	UF : 0, UT : 6,		CONFIG : 'N U T, 0, 0, 0',
	X =  237.113  mm,	Y =   -360.782  mm,	Z =   -247.837  mm,
	W =  90.000 deg,	P =   -89.765 deg,	R =   30.000 deg
};
P[393]{
   GP1:
	UF : 0, UT : 6,		CONFIG : 'N U T, 0, 0, 0',
	X =  236.281  mm,	Y =   -361.266  mm,	Z =   -247.891  mm,
	W =  90.000 deg,	P =   -89.765 deg,	R =   30.000 deg
};
P[394]{
   GP1:
	UF : 0, UT : 6,		CONFIG : 'N U T, 0, 0, 0',
	X =  236.253  mm,	Y =   -361.209  mm,	Z =   -246.975  mm,
	W =  90.000 deg,	P =   -89.765 deg,	R =   30.000 deg
};
P[395]{
   GP1:
	UF : 0, UT : 6,		CONFIG : 'N U T, 0, 0, 0',
	X =  235.670  mm,	Y =   -361.621  mm,	Z =   -247.913  mm,
	W =  90.000 deg,	P =   -89.765 deg,	R =   30.000 deg
};
P[396]{
   GP1:
	UF : 0, UT : 6,		CONFIG : 'N U T, 0, 0, 0',
	X =  235.399  mm,	Y =   -361.776  mm,	Z =   -247.895  mm,
	W =  90.000 deg,	P =   -89.765 deg,	R =   30.000 deg
};
P[397]{
   GP1:
	UF : 0, UT : 6,		CONFIG : 'N U T, 0, 0, 0',
	X =  234.392  mm,	Y =   -360.505  mm,	Z =   -224.946  mm,
	W =  90.000 deg,	P =   -89.765 deg,	R =   30.000 deg
};
P[398]{
   GP1:
	UF : 0, UT : 6,		CONFIG : 'N U T, 0, 0, 0',
	X =  234.357  mm,	Y =   -360.593  mm,	Z =   -225.785  mm,
	W =  90.000 deg,	P =   -89.765 deg,	R =   30.000 deg
};
P[399]{
   GP1:
	UF : 0, UT : 6,		CONFIG : 'N U T, 0, 0, 0',
	X =  234.000  mm,	Y =   -360.802  mm,	Z =   -225.822  mm,
	W =  90.000 deg,	P =   -89.765 deg,	R =   30.000 deg
};
P[400]{
   GP1:
	UF : 0, UT : 6,		CONFIG : 'N U T, 0, 0, 0',
	X =  233.702  mm,	Y =   -360.970  mm,	Z =   -225.770  mm,
	W =  90.000 deg,	P =   -89.765 deg,	R =   30.000 deg
};
P[401]{
   GP1:
	UF : 0, UT : 6,		CONFIG : 'N U T, 0, 0, 0',
	X =  233.487  mm,	Y =   -361.098  mm,	Z =   -225.822  mm,
	W =  90.000 deg,	P =   -89.765 deg,	R =   30.000 deg
};
P[402]{
   GP1:
	UF : 0, UT : 6,		CONFIG : 'N U T, 0, 0, 0',
	X =  233.404  mm,	Y =   -361.075  mm,	Z =   -224.940  mm,
	W =  90.000 deg,	P =   -89.765 deg,	R =   30.000 deg
};
P[403]{
   GP1:
	UF : 0, UT : 6,		CONFIG : 'N U T, 0, 0, 0',
	X =  232.811  mm,	Y =   -361.483  mm,	Z =   -225.762  mm,
	W =  90.000 deg,	P =   -89.765 deg,	R =   30.000 deg
};
P[404]{
   GP1:
	UF : 0, UT : 6,		CONFIG : 'N U T, 0, 0, 0',
	X =  232.580  mm,	Y =   -361.587  mm,	Z =   -225.392  mm,
	W =  90.000 deg,	P =   -89.765 deg,	R =   30.000 deg
};
P[405]{
   GP1:
	UF : 0, UT : 6,		CONFIG : 'N U T, 0, 0, 0',
	X =  232.529  mm,	Y =   -361.658  mm,	Z =   -225.909  mm,
	W =  90.000 deg,	P =   -89.765 deg,	R =   30.000 deg
};
P[406]{
   GP1:
	UF : 0, UT : 6,		CONFIG : 'N U T, 0, 0, 0',
	X =  232.294  mm,	Y =   -361.754  mm,	Z =   -225.413  mm,
	W =  90.000 deg,	P =   -89.765 deg,	R =   30.000 deg
};
P[407]{
   GP1:
	UF : 0, UT : 6,		CONFIG : 'N U T, 0, 0, 0',
	X =  232.210  mm,	Y =   -361.841  mm,	Z =   -225.896  mm,
	W =  90.000 deg,	P =   -89.765 deg,	R =   30.000 deg
};
P[408]{
   GP1:
	UF : 0, UT : 6,		CONFIG : 'N U T, 0, 0, 0',
	X =  231.623  mm,	Y =   -362.182  mm,	Z =   -225.911  mm,
	W =  90.000 deg,	P =   -89.765 deg,	R =   30.000 deg
};
P[409]{
   GP1:
	UF : 0, UT : 6,		CONFIG : 'N U T, 0, 0, 0',
	X =  231.557  mm,	Y =   -362.142  mm,	Z =   -224.952  mm,
	W =  90.000 deg,	P =   -89.765 deg,	R =   30.000 deg
};
P[410]{
   GP1:
	UF : 0, UT : 6,		CONFIG : 'N U T, 0, 0, 0',
	X =  231.491  mm,	Y =   -362.215  mm,	Z =   -225.396  mm,
	W =  90.000 deg,	P =   -89.765 deg,	R =   30.000 deg
};
P[411]{
   GP1:
	UF : 0, UT : 6,		CONFIG : 'N U T, 0, 0, 0',
	X =  231.269  mm,	Y =   -362.315  mm,	Z =   -225.031  mm,
	W =  90.000 deg,	P =   -89.765 deg,	R =   30.000 deg
};
P[412]{
   GP1:
	UF : 0, UT : 6,		CONFIG : 'N U T, 0, 0, 0',
	X =  231.297  mm,	Y =   -362.369  mm,	Z =   -225.901  mm,
	W =  90.000 deg,	P =   -89.765 deg,	R =   30.000 deg
};
P[413]{
   GP1:
	UF : 0, UT : 6,		CONFIG : 'N U T, 0, 0, 0',
	X =  230.990  mm,	Y =   -362.547  mm,	Z =   -225.923  mm,
	W =  90.000 deg,	P =   -89.765 deg,	R =   30.000 deg
};
P[414]{
   GP1:
	UF : 0, UT : 6,		CONFIG : 'N U T, 0, 0, 0',
	X =  230.655  mm,	Y =   -362.675  mm,	Z =   -225.107  mm,
	W =  90.000 deg,	P =   -89.765 deg,	R =   30.000 deg
};
P[415]{
   GP1:
	UF : 0, UT : 6,		CONFIG : 'N U T, 0, 0, 0',
	X =  230.373  mm,	Y =   -362.893  mm,	Z =   -225.776  mm,
	W =  90.000 deg,	P =   -89.765 deg,	R =   30.000 deg
};
P[416]{
   GP1:
	UF : 0, UT : 6,		CONFIG : 'N U T, 0, 0, 0',
	X =  229.910  mm,	Y =   -363.127  mm,	Z =   -225.378  mm,
	W =  90.000 deg,	P =   -89.765 deg,	R =   30.000 deg
};
P[417]{
   GP1:
	UF : 0, UT : 6,		CONFIG : 'N U T, 0, 0, 0',
	X =  229.140  mm,	Y =   -363.606  mm,	Z =   -225.794  mm,
	W =  90.000 deg,	P =   -89.765 deg,	R =   30.000 deg
};
P[418]{
   GP1:
	UF : 0, UT : 6,		CONFIG : 'N U T, 0, 0, 0',
	X =  228.874  mm,	Y =   -363.726  mm,	Z =   -225.370  mm,
	W =  90.000 deg,	P =   -89.765 deg,	R =   30.000 deg
};
P[419]{
   GP1:
	UF : 0, UT : 6,		CONFIG : 'N U T, 0, 0, 0',
	X =  228.845  mm,	Y =   -363.780  mm,	Z =   -225.848  mm,
	W =  90.000 deg,	P =   -89.765 deg,	R =   30.000 deg
};
P[420]{
   GP1:
	UF : 0, UT : 6,		CONFIG : 'N U T, 0, 0, 0',
	X =  227.859  mm,	Y =   -364.284  mm,	Z =   -225.040  mm,
	W =  90.000 deg,	P =   -89.765 deg,	R =   30.000 deg
};
P[421]{
   GP1:
	UF : 0, UT : 6,		CONFIG : 'N U T, 0, 0, 0',
	X =  227.784  mm,	Y =   -364.357  mm,	Z =   -225.398  mm,
	W =  90.000 deg,	P =   -89.765 deg,	R =   30.000 deg
};
P[422]{
   GP1:
	UF : 0, UT : 6,		CONFIG : 'N U T, 0, 0, 0',
	X =  227.246  mm,	Y =   -364.630  mm,	Z =   -224.931  mm,
	W =  90.000 deg,	P =   -89.765 deg,	R =   30.000 deg
};
P[423]{
   GP1:
	UF : 0, UT : 6,		CONFIG : 'N U T, 0, 0, 0',
	X =  227.248  mm,	Y =   -364.668  mm,	Z =   -225.413  mm,
	W =  90.000 deg,	P =   -89.765 deg,	R =   30.000 deg
};
P[424]{
   GP1:
	UF : 0, UT : 6,		CONFIG : 'N U T, 0, 0, 0',
	X =  226.957  mm,	Y =   -364.870  mm,	Z =   -225.849  mm,
	W =  90.000 deg,	P =   -89.765 deg,	R =   30.000 deg
};
P[425]{
   GP1:
	UF : 0, UT : 6,		CONFIG : 'N U T, 0, 0, 0',
	X =  226.306  mm,	Y =   -365.173  mm,	Z =   -224.949  mm,
	W =  90.000 deg,	P =   -89.765 deg,	R =   30.000 deg
};
P[426]{
   GP1:
	UF : 0, UT : 6,		CONFIG : 'N U T, 0, 0, 0',
	X =  226.123  mm,	Y =   -365.346  mm,	Z =   -225.786  mm,
	W =  90.000 deg,	P =   -89.765 deg,	R =   30.000 deg
};
P[427]{
   GP1:
	UF : 0, UT : 6,		CONFIG : 'N U T, 0, 0, 0',
	X =  225.718  mm,	Y =   -365.520  mm,	Z =   -225.031  mm,
	W =  90.000 deg,	P =   -89.765 deg,	R =   30.000 deg
};
P[428]{
   GP1:
	UF : 0, UT : 6,		CONFIG : 'N U T, 0, 0, 0',
	X =  225.480  mm,	Y =   -365.726  mm,	Z =   -225.890  mm,
	W =  90.000 deg,	P =   -89.765 deg,	R =   30.000 deg
};
P[429]{
   GP1:
	UF : 0, UT : 6,		CONFIG : 'N U T, 0, 0, 0',
	X =  225.376  mm,	Y =   -365.713  mm,	Z =   -224.981  mm,
	W =  90.000 deg,	P =   -89.765 deg,	R =   30.000 deg
};
P[430]{
   GP1:
	UF : 0, UT : 6,		CONFIG : 'N U T, 0, 0, 0',
	X =  225.172  mm,	Y =   -365.903  mm,	Z =   -225.869  mm,
	W =  90.000 deg,	P =   -89.765 deg,	R =   30.000 deg
};
P[431]{
   GP1:
	UF : 0, UT : 6,		CONFIG : 'N U T, 0, 0, 0',
	X =  224.799  mm,	Y =   -366.046  mm,	Z =   -224.974  mm,
	W =  90.000 deg,	P =   -89.765 deg,	R =   30.000 deg
};
P[432]{
   GP1:
	UF : 0, UT : 6,		CONFIG : 'N U T, 0, 0, 0',
	X =  224.881  mm,	Y =   -366.070  mm,	Z =   -225.869  mm,
	W =  90.000 deg,	P =   -89.765 deg,	R =   30.000 deg
};
P[433]{
   GP1:
	UF : 0, UT : 6,		CONFIG : 'N U T, 0, 0, 0',
	X =  224.484  mm,	Y =   -366.225  mm,	Z =   -224.935  mm,
	W =  90.000 deg,	P =   -89.765 deg,	R =   30.000 deg
};
P[434]{
   GP1:
	UF : 0, UT : 6,		CONFIG : 'N U T, 0, 0, 0',
	X =  223.897  mm,	Y =   -366.567  mm,	Z =   -224.985  mm,
	W =  90.000 deg,	P =   -89.765 deg,	R =   30.000 deg
};
P[435]{
   GP1:
	UF : 0, UT : 6,		CONFIG : 'N U T, 0, 0, 0',
	X =  223.958  mm,	Y =   -366.608  mm,	Z =   -225.921  mm,
	W =  90.000 deg,	P =   -89.765 deg,	R =   30.000 deg
};
P[436]{
   GP1:
	UF : 0, UT : 6,		CONFIG : 'N U T, 0, 0, 0',
	X =  223.659  mm,	Y =   -366.774  mm,	Z =   -225.845  mm,
	W =  90.000 deg,	P =   -89.765 deg,	R =   30.000 deg
};
P[437]{
   GP1:
	UF : 0, UT : 6,		CONFIG : 'N U T, 0, 0, 0',
	X =  223.279  mm,	Y =   -366.933  mm,	Z =   -225.088  mm,
	W =  90.000 deg,	P =   -89.765 deg,	R =   30.000 deg
};
P[438]{
   GP1:
	UF : 0, UT : 6,		CONFIG : 'N U T, 0, 0, 0',
	X =  222.812  mm,	Y =   -367.228  mm,	Z =   -225.404  mm,
	W =  90.000 deg,	P =   -89.765 deg,	R =   30.000 deg
};
P[439]{
   GP1:
	UF : 0, UT : 6,		CONFIG : 'N U T, 0, 0, 0',
	X =  222.634  mm,	Y =   -367.307  mm,	Z =   -225.106  mm,
	W =  90.000 deg,	P =   -89.765 deg,	R =   30.000 deg
};
P[440]{
   GP1:
	UF : 0, UT : 6,		CONFIG : 'N U T, 0, 0, 0',
	X =  222.336  mm,	Y =   -367.475  mm,	Z =   -225.055  mm,
	W =  90.000 deg,	P =   -89.765 deg,	R =   30.000 deg
};
P[441]{
   GP1:
	UF : 0, UT : 6,		CONFIG : 'N U T, 0, 0, 0',
	X =  222.421  mm,	Y =   -367.495  mm,	Z =   -225.924  mm,
	W =  90.000 deg,	P =   -89.765 deg,	R =   30.000 deg
};
P[442]{
   GP1:
	UF : 0, UT : 6,		CONFIG : 'N U T, 0, 0, 0',
	X =  222.156  mm,	Y =   -367.606  mm,	Z =   -225.402  mm,
	W =  90.000 deg,	P =   -89.765 deg,	R =   30.000 deg
};
P[443]{
   GP1:
	UF : 0, UT : 6,		CONFIG : 'N U T, 0, 0, 0',
	X =  222.101  mm,	Y =   -367.678  mm,	Z =   -225.899  mm,
	W =  90.000 deg,	P =   -89.765 deg,	R =   30.000 deg
};
P[444]{
   GP1:
	UF : 0, UT : 6,		CONFIG : 'N U T, 0, 0, 0',
	X =  221.716  mm,	Y =   -367.828  mm,	Z =   -224.998  mm,
	W =  90.000 deg,	P =   -89.765 deg,	R =   30.000 deg
};
P[445]{
   GP1:
	UF : 0, UT : 6,		CONFIG : 'N U T, 0, 0, 0',
	X =  221.807  mm,	Y =   -367.841  mm,	Z =   -225.809  mm,
	W =  90.000 deg,	P =   -89.765 deg,	R =   30.000 deg
};
P[446]{
   GP1:
	UF : 0, UT : 6,		CONFIG : 'N U T, 0, 0, 0',
	X =  221.506  mm,	Y =   -368.013  mm,	Z =   -225.782  mm,
	W =  90.000 deg,	P =   -89.765 deg,	R =   30.000 deg
};
P[447]{
   GP1:
	UF : 0, UT : 6,		CONFIG : 'N U T, 0, 0, 0',
	X =  221.122  mm,	Y =   -368.170  mm,	Z =   -224.979  mm,
	W =  90.000 deg,	P =   -89.765 deg,	R =   30.000 deg
};
P[448]{
   GP1:
	UF : 0, UT : 6,		CONFIG : 'N U T, 0, 0, 0',
	X =  220.843  mm,	Y =   -368.401  mm,	Z =   -225.860  mm,
	W =  90.000 deg,	P =   -89.765 deg,	R =   30.000 deg
};
P[449]{
   GP1:
	UF : 0, UT : 6,		CONFIG : 'N U T, 0, 0, 0',
	X =  220.507  mm,	Y =   -368.525  mm,	Z =   -224.981  mm,
	W =  90.000 deg,	P =   -89.765 deg,	R =   30.000 deg
};
P[450]{
   GP1:
	UF : 0, UT : 6,		CONFIG : 'N U T, 0, 0, 0',
	X =  220.223  mm,	Y =   -368.756  mm,	Z =   -225.819  mm,
	W =  90.000 deg,	P =   -89.765 deg,	R =   30.000 deg
};
P[451]{
   GP1:
	UF : 0, UT : 6,		CONFIG : 'N U T, 0, 0, 0',
	X =  219.902  mm,	Y =   -368.872  mm,	Z =   -224.956  mm,
	W =  90.000 deg,	P =   -89.765 deg,	R =   30.000 deg
};
P[452]{
   GP1:
	UF : 0, UT : 6,		CONFIG : 'N U T, 0, 0, 0',
	X =  219.585  mm,	Y =   -369.089  mm,	Z =   -225.369  mm,
	W =  90.000 deg,	P =   -89.765 deg,	R =   30.000 deg
};
P[453]{
   GP1:
	UF : 0, UT : 6,		CONFIG : 'N U T, 0, 0, 0',
	X =  219.644  mm,	Y =   -369.097  mm,	Z =   -225.904  mm,
	W =  90.000 deg,	P =   -89.765 deg,	R =   30.000 deg
};
P[454]{
   GP1:
	UF : 0, UT : 6,		CONFIG : 'N U T, 0, 0, 0',
	X =  219.320  mm,	Y =   -369.278  mm,	Z =   -225.830  mm,
	W =  90.000 deg,	P =   -89.765 deg,	R =   30.000 deg
};
P[455]{
   GP1:
	UF : 0, UT : 6,		CONFIG : 'N U T, 0, 0, 0',
	X =  218.586  mm,	Y =   -369.630  mm,	Z =   -224.926  mm,
	W =  90.000 deg,	P =   -89.765 deg,	R =   30.000 deg
};
P[456]{
   GP1:
	UF : 0, UT : 6,		CONFIG : 'N U T, 0, 0, 0',
	X =  218.442  mm,	Y =   -369.788  mm,	Z =   -225.856  mm,
	W =  90.000 deg,	P =   -89.765 deg,	R =   30.000 deg
};
P[457]{
   GP1:
	UF : 0, UT : 6,		CONFIG : 'N U T, 0, 0, 0',
	X =  217.955  mm,	Y =   -370.032  mm,	Z =   -225.398  mm,
	W =  90.000 deg,	P =   -89.765 deg,	R =   30.000 deg
};
P[458]{
   GP1:
	UF : 0, UT : 6,		CONFIG : 'N U T, 0, 0, 0',
	X =  217.837  mm,	Y =   -370.100  mm,	Z =   -225.400  mm,
	W =  90.000 deg,	P =   -89.765 deg,	R =   30.000 deg
};
P[459]{
   GP1:
	UF : 0, UT : 6,		CONFIG : 'N U T, 0, 0, 0',
	X =  217.794  mm,	Y =   -370.161  mm,	Z =   -225.844  mm,
	W =  90.000 deg,	P =   -89.765 deg,	R =   30.000 deg
};
P[460]{
   GP1:
	UF : 0, UT : 6,		CONFIG : 'N U T, 0, 0, 0',
	X =  217.511  mm,	Y =   -370.286  mm,	Z =   -225.369  mm,
	W =  90.000 deg,	P =   -89.765 deg,	R =   30.000 deg
};
P[461]{
   GP1:
	UF : 0, UT : 6,		CONFIG : 'N U T, 0, 0, 0',
	X =  217.487  mm,	Y =   -370.338  mm,	Z =   -225.839  mm,
	W =  90.000 deg,	P =   -89.765 deg,	R =   30.000 deg
};
P[462]{
   GP1:
	UF : 0, UT : 6,		CONFIG : 'N U T, 0, 0, 0',
	X =  217.210  mm,	Y =   -370.501  mm,	Z =   -225.878  mm,
	W =  90.000 deg,	P =   -89.765 deg,	R =   30.000 deg
};
P[463]{
   GP1:
	UF : 0, UT : 6,		CONFIG : 'N U T, 0, 0, 0',
	X =  216.778  mm,	Y =   -370.682  mm,	Z =   -225.031  mm,
	W =  90.000 deg,	P =   -89.765 deg,	R =   30.000 deg
};
P[464]{
   GP1:
	UF : 0, UT : 6,		CONFIG : 'N U T, 0, 0, 0',
	X =  216.880  mm,	Y =   -370.686  mm,	Z =   -225.816  mm,
	W =  90.000 deg,	P =   -89.765 deg,	R =   30.000 deg
};
P[465]{
   GP1:
	UF : 0, UT : 6,		CONFIG : 'N U T, 0, 0, 0',
	X =  216.154  mm,	Y =   -371.071  mm,	Z =   -225.383  mm,
	W =  90.000 deg,	P =   -89.765 deg,	R =   30.000 deg
};
P[466]{
   GP1:
	UF : 0, UT : 6,		CONFIG : 'N U T, 0, 0, 0',
	X =  215.904  mm,	Y =   -371.214  mm,	Z =   -225.372  mm,
	W =  90.000 deg,	P =   -89.765 deg,	R =   30.000 deg
};
P[467]{
   GP1:
	UF : 0, UT : 6,		CONFIG : 'N U T, 0, 0, 0',
	X =  215.958  mm,	Y =   -371.227  mm,	Z =   -225.918  mm,
	W =  90.000 deg,	P =   -89.765 deg,	R =   30.000 deg
};
P[468]{
   GP1:
	UF : 0, UT : 6,		CONFIG : 'N U T, 0, 0, 0',
	X =  215.665  mm,	Y =   -371.387  mm,	Z =   -225.804  mm,
	W =  90.000 deg,	P =   -89.765 deg,	R =   30.000 deg
};
P[469]{
   GP1:
	UF : 0, UT : 6,		CONFIG : 'N U T, 0, 0, 0',
	X =  215.331  mm,	Y =   -371.586  mm,	Z =   -225.886  mm,
	W =  90.000 deg,	P =   -89.765 deg,	R =   30.000 deg
};
P[470]{
   GP1:
	UF : 0, UT : 6,		CONFIG : 'N U T, 0, 0, 0',
	X =  215.026  mm,	Y =   -371.742  mm,	Z =   -225.177  mm,
	W =  90.000 deg,	P =   -89.765 deg,	R =   30.000 deg
};
P[471]{
   GP1:
	UF : 0, UT : 6,		CONFIG : 'N U T, 0, 0, 0',
	X =  215.096  mm,	Y =   -371.773  mm,	Z =   -225.898  mm,
	W =  90.000 deg,	P =   -89.765 deg,	R =   30.000 deg
};
P[472]{
   GP1:
	UF : 0, UT : 6,		CONFIG : 'N U T, 0, 0, 0',
	X =  215.157  mm,	Y =   -372.393  mm,	Z =   -224.958  mm,
	W =  90.000 deg,	P =   -89.765 deg,	R =   30.000 deg
};
P[473]{
   GP1:
	UF : 0, UT : 6,		CONFIG : 'N U T, 0, 0, 0',
	X =  215.297  mm,	Y =   -372.394  mm,	Z =   -225.902  mm,
	W =  90.000 deg,	P =   -89.765 deg,	R =   30.000 deg
};
P[474]{
   GP1:
	UF : 0, UT : 6,		CONFIG : 'N U T, 0, 0, 0',
	X =  215.529  mm,	Y =   -372.532  mm,	Z =   -225.806  mm,
	W =  90.000 deg,	P =   -89.765 deg,	R =   30.000 deg
};
P[475]{
   GP1:
	UF : 0, UT : 6,		CONFIG : 'N U T, 0, 0, 0',
	X =  215.945  mm,	Y =   -372.668  mm,	Z =   -225.782  mm,
	W =  90.000 deg,	P =   -89.765 deg,	R =   30.000 deg
};
P[476]{
   GP1:
	UF : 0, UT : 6,		CONFIG : 'N U T, 0, 0, 0',
	X =  187.636  mm,	Y =   -376.299  mm,	Z =   -225.905  mm,
	W =  179.765 deg,	P =   0.000 deg,	R =   30.000 deg
};
P[477]{
   GP1:
	UF : 0, UT : 6,		CONFIG : 'N U T, 0, 0, 0',
	X =  187.516  mm,	Y =   -376.334  mm,	Z =   -225.076  mm,
	W =  179.765 deg,	P =   0.000 deg,	R =   30.000 deg
};
P[478]{
   GP1:
	UF : 0, UT : 6,		CONFIG : 'N U T, 0, 0, 0',
	X =  186.272  mm,	Y =   -378.286  mm,	Z =   -224.926  mm,
	W =  179.765 deg,	P =   0.000 deg,	R =   30.000 deg
};
P[479]{
   GP1:
	UF : 0, UT : 6,		CONFIG : 'N U T, 0, 0, 0',
	X =  186.053  mm,	Y =   -379.156  mm,	Z =   -225.859  mm,
	W =  179.765 deg,	P =   0.000 deg,	R =   30.000 deg
};
P[480]{
   GP1:
	UF : 0, UT : 6,		CONFIG : 'N U T, 0, 0, 0',
	X =  185.851  mm,	Y =   -379.926  mm,	Z =   -225.382  mm,
	W =  179.765 deg,	P =   0.000 deg,	R =   30.000 deg
};
P[481]{
   GP1:
	UF : 0, UT : 6,		CONFIG : 'N U T, 0, 0, 0',
	X =  185.800  mm,	Y =   -380.295  mm,	Z =   -225.483  mm,
	W =  179.765 deg,	P =   0.000 deg,	R =   30.000 deg
};
P[482]{
   GP1:
	UF : 0, UT : 6,		CONFIG : 'N U T, 0, 0, 0',
	X =  185.847  mm,	Y =   -380.797  mm,	Z =   -225.872  mm,
	W =  179.765 deg,	P =   0.000 deg,	R =   30.000 deg
};
P[483]{
   GP1:
	UF : 0, UT : 6,		CONFIG : 'N U T, 0, 0, 0',
	X =  185.769  mm,	Y =   -380.859  mm,	Z =   -224.974  mm,
	W =  179.765 deg,	P =   0.000 deg,	R =   30.000 deg
};
P[484]{
   GP1:
	UF : 0, UT : 6,		CONFIG : 'N U T, 0, 0, 0',
	X =  185.896  mm,	Y =   -381.491  mm,	Z =   -225.879  mm,
	W =  179.765 deg,	P =   0.000 deg,	R =   30.000 deg
};
P[485]{
   GP1:
	UF : 0, UT : 6,		CONFIG : 'N U T, 0, 0, 0',
	X =  186.008  mm,	Y =   -382.255  mm,	Z =   -225.033  mm,
	W =  179.765 deg,	P =   0.000 deg,	R =   30.000 deg
};
P[486]{
   GP1:
	UF : 0, UT : 6,		CONFIG : 'N U T, 0, 0, 0',
	X =  186.228  mm,	Y =   -382.820  mm,	Z =   -224.959  mm,
	W =  179.765 deg,	P =   0.000 deg,	R =   30.000 deg
};
P[487]{
   GP1:
	UF : 0, UT : 6,		CONFIG : 'N U T, 0, 0, 0',
	X =  186.619  mm,	Y =   -383.588  mm,	Z =   -225.001  mm,
	W =  179.765 deg,	P =   0.000 deg,	R =   30.000 deg
};
P[488]{
   GP1:
	UF : 0, UT : 6,		CONFIG : 'N U T, 0, 0, 0',
	X =  186.703  mm,	Y =   -383.610  mm,	Z =   -225.898  mm,
	W =  179.765 deg,	P =   0.000 deg,	R =   30.000 deg
};
P[489]{
   GP1:
	UF : 0, UT : 6,		CONFIG : 'N U T, 0, 0, 0',
	X =  187.014  mm,	Y =   -384.264  mm,	Z =   -225.061  mm,
	W =  179.765 deg,	P =   0.000 deg,	R =   30.000 deg
};
P[490]{
   GP1:
	UF : 0, UT : 6,		CONFIG : 'N U T, 0, 0, 0',
	X =  187.375  mm,	Y =   -384.782  mm,	Z =   -225.838  mm,
	W =  179.765 deg,	P =   0.000 deg,	R =   30.000 deg
};
P[491]{
   GP1:
	UF : 0, UT : 6,		CONFIG : 'N U T, 0, 0, 0',
	X =  187.642  mm,	Y =   -385.308  mm,	Z =   -225.374  mm,
	W =  179.765 deg,	P =   0.000 deg,	R =   30.000 deg
};
P[492]{
   GP1:
	UF : 0, UT : 6,		CONFIG : 'N U T, 0, 0, 0',
	X =  188.498  mm,	Y =   -386.785  mm,	Z =   -225.413  mm,
	W =  179.765 deg,	P =   0.000 deg,	R =   30.000 deg
};
P[493]{
   GP1:
	UF : 0, UT : 6,		CONFIG : 'N U T, 0, 0, 0',
	X =  188.473  mm,	Y =   -386.803  mm,	Z =   -224.982  mm,
	W =  179.765 deg,	P =   0.000 deg,	R =   30.000 deg
};
P[494]{
   GP1:
	UF : 0, UT : 6,		CONFIG : 'N U T, 0, 0, 0',
	X =  188.877  mm,	Y =   -387.392  mm,	Z =   -225.780  mm,
	W =  179.765 deg,	P =   0.000 deg,	R =   30.000 deg
};
P[495]{
   GP1:
	UF : 0, UT : 6,		CONFIG : 'N U T, 0, 0, 0',
	X =  189.626  mm,	Y =   -388.676  mm,	Z =   -225.866  mm,
	W =  179.765 deg,	P =   0.000 deg,	R =   30.000 deg
};
P[496]{
   GP1:
	UF : 0, UT : 6,		CONFIG : 'N U T, 0, 0, 0',
	X =  190.032  mm,	Y =   -389.448  mm,	Z =   -225.376  mm,
	W =  179.765 deg,	P =   0.000 deg,	R =   30.000 deg
};
P[497]{
   GP1:
	UF : 0, UT : 6,		CONFIG : 'N U T, 0, 0, 0',
	X =  190.306  mm,	Y =   -389.869  mm,	Z =   -225.756  mm,
	W =  179.765 deg,	P =   0.000 deg,	R =   30.000 deg
};
P[498]{
   GP1:
	UF : 0, UT : 6,		CONFIG : 'N U T, 0, 0, 0',
	X =  191.062  mm,	Y =   -391.232  mm,	Z =   -225.376  mm,
	W =  179.765 deg,	P =   0.000 deg,	R =   30.000 deg
};
P[499]{
   GP1:
	UF : 0, UT : 6,		CONFIG : 'N U T, 0, 0, 0',
	X =  191.772  mm,	Y =   -392.386  mm,	Z =   -225.912  mm,
	W =  179.765 deg,	P =   0.000 deg,	R =   30.000 deg
};
P[500]{
   GP1:
	UF : 0, UT : 6,		CONFIG : 'N U T, 0, 0, 0',
	X =  191.716  mm,	Y =   -392.426  mm,	Z =   -224.935  mm,
	W =  179.765 deg,	P =   0.000 deg,	R =   30.000 deg
};
P[501]{
   GP1:
	UF : 0, UT : 6,		CONFIG : 'N U T, 0, 0, 0',
	X =  192.126  mm,	Y =   -393.072  mm,	Z =   -225.383  mm,
	W =  179.765 deg,	P =   0.000 deg,	R =   30.000 deg
};
P[502]{
   GP1:
	UF : 0, UT : 6,		CONFIG : 'N U T, 0, 0, 0',
	X =  192.449  mm,	Y =   -393.561  mm,	Z =   -225.890  mm,
	W =  179.765 deg,	P =   0.000 deg,	R =   30.000 deg
};
P[503]{
   GP1:
	UF : 0, UT : 6,		CONFIG : 'N U T, 0, 0, 0',
	X =  192.468  mm,	Y =   -393.712  mm,	Z =   -225.051  mm,
	W =  179.765 deg,	P =   0.000 deg,	R =   30.000 deg
};
P[504]{
   GP1:
	UF : 0, UT : 6,		CONFIG : 'N U T, 0, 0, 0',
	X =  193.110  mm,	Y =   -394.836  mm,	Z =   -224.967  mm,
	W =  179.765 deg,	P =   0.000 deg,	R =   30.000 deg
};
P[505]{
   GP1:
	UF : 0, UT : 6,		CONFIG : 'N U T, 0, 0, 0',
	X =  193.212  mm,	Y =   -394.888  mm,	Z =   -225.862  mm,
	W =  179.765 deg,	P =   0.000 deg,	R =   30.000 deg
};
P[506]{
   GP1:
	UF : 0, UT : 6,		CONFIG : 'N U T, 0, 0, 0',
	X =  193.527  mm,	Y =   -395.560  mm,	Z =   -224.953  mm,
	W =  179.765 deg,	P =   0.000 deg,	R =   30.000 deg
};
P[507]{
   GP1:
	UF : 0, UT : 6,		CONFIG : 'N U T, 0, 0, 0',
	X =  194.305  mm,	Y =   -396.776  mm,	Z =   -225.891  mm,
	W =  179.765 deg,	P =   0.000 deg,	R =   30.000 deg
};
P[508]{
   GP1:
	UF : 0, UT : 6,		CONFIG : 'N U T, 0, 0, 0',
	X =  194.425  mm,	Y =   -397.052  mm,	Z =   -225.405  mm,
	W =  179.765 deg,	P =   0.000 deg,	R =   30.000 deg
};
P[509]{
   GP1:
	UF : 0, UT : 6,		CONFIG : 'N U T, 0, 0, 0',
	X =  194.620  mm,	Y =   -397.452  mm,	Z =   -224.964  mm,
	W =  179.765 deg,	P =   0.000 deg,	R =   30.000 deg
};
P[510]{
   GP1:
	UF : 0, UT : 6,		CONFIG : 'N U T, 0, 0, 0',
	X =  194.695  mm,	Y =   -397.452  mm,	Z =   -225.885  mm,
	W =  179.765 deg,	P =   0.000 deg,	R =   30.000 deg
};
P[511]{
   GP1:
	UF : 0, UT : 6,		CONFIG : 'N U T, 0, 0, 0',
	X =  194.972  mm,	Y =   -398.059  mm,	Z =   -224.972  mm,
	W =  179.765 deg,	P =   0.000 deg,	R =   30.000 deg
};
P[512]{
   GP1:
	UF : 0, UT : 6,		CONFIG : 'N U T, 0, 0, 0',
	X =  195.239  mm,	Y =   -398.464  mm,	Z =   -225.395  mm,
	W =  179.765 deg,	P =   0.000 deg,	R =   30.000 deg
};
P[513]{
   GP1:
	UF : 0, UT : 6,		CONFIG : 'N U T, 0, 0, 0',
	X =  195.836  mm,	Y =   -399.432  mm,	Z =   -225.860  mm,
	W =  179.765 deg,	P =   0.000 deg,	R =   30.000 deg
};
P[514]{
   GP1:
	UF : 0, UT : 6,		CONFIG : 'N U T, 0, 0, 0',
	X =  195.979  mm,	Y =   -399.749  mm,	Z =   -225.363  mm,
	W =  179.765 deg,	P =   0.000 deg,	R =   30.000 deg
};
P[515]{
   GP1:
	UF : 0, UT : 6,		CONFIG : 'N U T, 0, 0, 0',
	X =  196.097  mm,	Y =   -400.011  mm,	Z =   -224.947  mm,
	W =  179.765 deg,	P =   0.000 deg,	R =   30.000 deg
};
P[516]{
   GP1:
	UF : 0, UT : 6,		CONFIG : 'N U T, 0, 0, 0',
	X =  196.178  mm,	Y =   -400.041  mm,	Z =   -225.740  mm,
	W =  179.765 deg,	P =   0.000 deg,	R =   30.000 deg
};
P[517]{
   GP1:
	UF : 0, UT : 6,		CONFIG : 'N U T, 0, 0, 0',
	X =  196.456  mm,	Y =   -400.527  mm,	Z =   -225.708  mm,
	W =  179.765 deg,	P =   0.000 deg,	R =   30.000 deg
};
P[518]{
   GP1:
	UF : 0, UT : 6,		CONFIG : 'N U T, 0, 0, 0',
	X =  196.993  mm,	Y =   -401.498  mm,	Z =   -225.413  mm,
	W =  179.765 deg,	P =   0.000 deg,	R =   30.000 deg
};
P[519]{
   GP1:
	UF : 0, UT : 6,		CONFIG : 'N U T, 0, 0, 0',
	X =  197.525  mm,	Y =   -402.479  mm,	Z =   -225.000  mm,
	W =  179.765 deg,	P =   0.000 deg,	R =   30.000 deg
};
P[520]{
   GP1:
	UF : 0, UT : 6,		CONFIG : 'N U T, 0, 0, 0',
	X =  197.618  mm,	Y =   -402.582  mm,	Z =   -225.399  mm,
	W =  179.765 deg,	P =   0.000 deg,	R =   30.000 deg
};
P[521]{
   GP1:
	UF : 0, UT : 6,		CONFIG : 'N U T, 0, 0, 0',
	X =  197.819  mm,	Y =   -402.997  mm,	Z =   -224.930  mm,
	W =  179.765 deg,	P =   0.000 deg,	R =   30.000 deg
};
P[522]{
   GP1:
	UF : 0, UT : 6,		CONFIG : 'N U T, 0, 0, 0',
	X =  198.007  mm,	Y =   -403.202  mm,	Z =   -225.792  mm,
	W =  179.765 deg,	P =   0.000 deg,	R =   30.000 deg
};
P[523]{
   GP1:
	UF : 0, UT : 6,		CONFIG : 'N U T, 0, 0, 0',
	X =  198.357  mm,	Y =   -403.809  mm,	Z =   -225.778  mm,
	W =  179.765 deg,	P =   0.000 deg,	R =   30.000 deg
};
P[524]{
   GP1:
	UF : 0, UT : 6,		CONFIG : 'N U T, 0, 0, 0',
	X =  198.596  mm,	Y =   -404.332  mm,	Z =   -225.007  mm,
	W =  179.765 deg,	P =   0.000 deg,	R =   30.000 deg
};
P[525]{
   GP1:
	UF : 0, UT : 6,		CONFIG : 'N U T, 0, 0, 0',
	X =  198.663  mm,	Y =   -404.328  mm,	Z =   -225.859  mm,
	W =  179.765 deg,	P =   0.000 deg,	R =   30.000 deg
};
P[526]{
   GP1:
	UF : 0, UT : 6,		CONFIG : 'N U T, 0, 0, 0',
	X =  199.022  mm,	Y =   -405.057  mm,	Z =   -225.090  mm,
	W =  179.765 deg,	P =   0.000 deg,	R =   30.000 deg
};
P[527]{
   GP1:
	UF : 0, UT : 6,		CONFIG : 'N U T, 0, 0, 0',
	X =  199.160  mm,	Y =   -405.255  mm,	Z =   -225.389  mm,
	W =  179.765 deg,	P =   0.000 deg,	R =   30.000 deg
};
P[528]{
   GP1:
	UF : 0, UT : 6,		CONFIG : 'N U T, 0, 0, 0',
	X =  199.411  mm,	Y =   -405.618  mm,	Z =   -225.906  mm,
	W =  179.765 deg,	P =   0.000 deg,	R =   30.000 deg
};
P[529]{
   GP1:
	UF : 0, UT : 6,		CONFIG : 'N U T, 0, 0, 0',
	X =  199.783  mm,	Y =   -406.278  mm,	Z =   -225.793  mm,
	W =  179.765 deg,	P =   0.000 deg,	R =   30.000 deg
};
P[530]{
   GP1:
	UF : 0, UT : 6,		CONFIG : 'N U T, 0, 0, 0',
	X =  200.163  mm,	Y =   -406.994  mm,	Z =   -225.381  mm,
	W =  179.765 deg,	P =   0.000 deg,	R =   30.000 deg
};
P[531]{
   GP1:
	UF : 0, UT : 6,		CONFIG : 'N U T, 0, 0, 0',
	X =  200.461  mm,	Y =   -407.455  mm,	Z =   -225.770  mm,
	W =  179.765 deg,	P =   0.000 deg,	R =   30.000 deg
};
P[532]{
   GP1:
	UF : 0, UT : 6,		CONFIG : 'N U T, 0, 0, 0',
	X =  200.460  mm,	Y =   -407.564  mm,	Z =   -224.979  mm,
	W =  179.765 deg,	P =   0.000 deg,	R =   30.000 deg
};
P[533]{
   GP1:
	UF : 0, UT : 6,		CONFIG : 'N U T, 0, 0, 0',
	X =  200.697  mm,	Y =   -407.920  mm,	Z =   -225.364  mm,
	W =  179.765 deg,	P =   0.000 deg,	R =   30.000 deg
};
P[534]{
   GP1:
	UF : 0, UT : 6,		CONFIG : 'N U T, 0, 0, 0',
	X =  200.853  mm,	Y =   -408.124  mm,	Z =   -225.829  mm,
	W =  179.765 deg,	P =   0.000 deg,	R =   30.000 deg
};
P[535]{
   GP1:
	UF : 0, UT : 6,		CONFIG : 'N U T, 0, 0, 0',
	X =  201.213  mm,	Y =   -408.809  mm,	Z =   -225.405  mm,
	W =  179.765 deg,	P =   0.000 deg,	R =   30.000 deg
};
P[536]{
   GP1:
	UF : 0, UT : 6,		CONFIG : 'N U T, 0, 0, 0',
	X =  201.559  mm,	Y =   -409.349  mm,	Z =   -225.819  mm,
	W =  179.765 deg,	P =   0.000 deg,	R =   30.000 deg
};
P[537]{
   GP1:
	UF : 0, UT : 6,		CONFIG : 'N U T, 0, 0, 0',
	X =  201.861  mm,	Y =   -409.821  mm,	Z =   -225.925  mm,
	W =  179.765 deg,	P =   0.000 deg,	R =   30.000 deg
};
P[538]{
   GP1:
	UF : 0, UT : 6,		CONFIG : 'N U T, 0, 0, 0',
	X =  201.962  mm,	Y =   -410.061  mm,	Z =   -225.152  mm,
	W =  179.765 deg,	P =   0.000 deg,	R =   30.000 deg
};
P[539]{
   GP1:
	UF : 0, UT : 6,		CONFIG : 'N U T, 0, 0, 0',
	X =  202.367  mm,	Y =   -410.521  mm,	Z =   -225.735  mm,
	W =  179.765 deg,	P =   0.000 deg,	R =   30.000 deg
};
P[540]{
   GP1:
	UF : 0, UT : 6,		CONFIG : 'N U T, 0, 0, 0',
	X =  204.004  mm,	Y =   -411.840  mm,	Z =   -224.989  mm,
	W =  179.765 deg,	P =   0.000 deg,	R =   30.000 deg
};
P[541]{
   GP1:
	UF : 0, UT : 6,		CONFIG : 'N U T, 0, 0, 0',
	X =  204.055  mm,	Y =   -411.791  mm,	Z =   -225.781  mm,
	W =  179.765 deg,	P =   0.000 deg,	R =   30.000 deg
};
P[542]{
   GP1:
	UF : 0, UT : 6,		CONFIG : 'N U T, 0, 0, 0',
	X =  204.385  mm,	Y =   -411.907  mm,	Z =   -225.877  mm,
	W =  179.765 deg,	P =   0.000 deg,	R =   30.000 deg
};
P[543]{
   GP1:
	UF : 0, UT : 6,		CONFIG : 'N U T, 0, 0, 0',
	X =  205.041  mm,	Y =   -412.216  mm,	Z =   -224.940  mm,
	W =  179.765 deg,	P =   0.000 deg,	R =   30.000 deg
};
P[544]{
   GP1:
	UF : 0, UT : 6,		CONFIG : 'N U T, 0, 0, 0',
	X =  206.124  mm,	Y =   -412.327  mm,	Z =   -225.830  mm,
	W =  179.765 deg,	P =   0.000 deg,	R =   30.000 deg
};
P[545]{
   GP1:
	UF : 0, UT : 6,		CONFIG : 'N U T, 0, 0, 0',
	X =  207.318  mm,	Y =   -412.345  mm,	Z =   -225.752  mm,
	W =  179.765 deg,	P =   0.000 deg,	R =   30.000 deg
};
P[546]{
   GP1:
	UF : 0, UT : 6,		CONFIG : 'N U T, 0, 0, 0',
	X =  208.519  mm,	Y =   -412.173  mm,	Z =   -225.881  mm,
	W =  179.765 deg,	P =   0.000 deg,	R =   30.000 deg
};
P[547]{
   GP1:
	UF : 0, UT : 6,		CONFIG : 'N U T, 0, 0, 0',
	X =  225.635  mm,	Y =   -389.642  mm,	Z =   -225.857  mm,
	W =  90.000 deg,	P =   89.765 deg,	R =   30.000 deg
};
P[548]{
   GP1:
	UF : 0, UT : 6,		CONFIG : 'N U T, 0, 0, 0',
	X =  225.559  mm,	Y =   -389.777  mm,	Z =   -224.931  mm,
	W =  90.000 deg,	P =   89.765 deg,	R =   30.000 deg
};
P[549]{
   GP1:
	UF : 0, UT : 6,		CONFIG : 'N U T, 0, 0, 0',
	X =  225.510  mm,	Y =   -390.047  mm,	Z =   -224.972  mm,
	W =  90.000 deg,	P =   89.765 deg,	R =   30.000 deg
};
P[550]{
   GP1:
	UF : 0, UT : 6,		CONFIG : 'N U T, 0, 0, 0',
	X =  225.570  mm,	Y =   -389.966  mm,	Z =   -225.847  mm,
	W =  90.000 deg,	P =   89.765 deg,	R =   30.000 deg
};
P[551]{
   GP1:
	UF : 0, UT : 6,		CONFIG : 'N U T, 0, 0, 0',
	X =  225.575  mm,	Y =   -390.248  mm,	Z =   -225.872  mm,
	W =  90.000 deg,	P =   89.765 deg,	R =   30.000 deg
};
P[552]{
   GP1:
	UF : 0, UT : 6,		CONFIG : 'N U T, 0, 0, 0',
	X =  225.642  mm,	Y =   -390.596  mm,	Z =   -225.749  mm,
	W =  90.000 deg,	P =   89.765 deg,	R =   30.000 deg
};
P[553]{
   GP1:
	UF : 0, UT : 6,		CONFIG : 'N U T, 0, 0, 0',
	X =  225.582  mm,	Y =   -390.691  mm,	Z =   -224.931  mm,
	W =  90.000 deg,	P =   89.765 deg,	R =   30.000 deg
};
P[554]{
   GP1:
	UF : 0, UT : 6,		CONFIG : 'N U T, 0, 0, 0',
	X =  225.755  mm,	Y =   -390.830  mm,	Z =   -224.945  mm,
	W =  90.000 deg,	P =   89.765 deg,	R =   30.000 deg
};
P[555]{
   GP1:
	UF : 0, UT : 6,		CONFIG : 'N U T, 0, 0, 0',
	X =  225.923  mm,	Y =   -390.794  mm,	Z =   -225.041  mm,
	W =  90.000 deg,	P =   89.765 deg,	R =   30.000 deg
};
P[556]{
   GP1:
	UF : 0, UT : 6,		CONFIG : 'N U T, 0, 0, 0',
	X =  226.292  mm,	Y =   -390.574  mm,	Z =   -225.872  mm,
	W =  90.000 deg,	P =   89.765 deg,	R =   30.000 deg
};
P[557]{
   GP1:
	UF : 0, UT : 6,		CONFIG : 'N U T, 0, 0, 0',
	X =  226.262  mm,	Y =   -390.660  mm,	Z =   -225.010  mm,
	W =  90.000 deg,	P =   89.765 deg,	R =   30.000 deg
};
P[558]{
   GP1:
	UF : 0, UT : 6,		CONFIG : 'N U T, 0, 0, 0',
	X =  226.648  mm,	Y =   -390.366  mm,	Z =   -225.894  mm,
	W =  90.000 deg,	P =   89.765 deg,	R =   30.000 deg
};
P[559]{
   GP1:
	UF : 0, UT : 6,		CONFIG : 'N U T, 0, 0, 0',
	X =  226.828  mm,	Y =   -390.309  mm,	Z =   -225.316  mm,
	W =  90.000 deg,	P =   89.765 deg,	R =   30.000 deg
};
P[560]{
   GP1:
	UF : 0, UT : 6,		CONFIG : 'N U T, 0, 0, 0',
	X =  226.929  mm,	Y =   -390.214  mm,	Z =   -225.768  mm,
	W =  90.000 deg,	P =   89.765 deg,	R =   30.000 deg
};
P[561]{
   GP1:
	UF : 0, UT : 6,		CONFIG : 'N U T, 0, 0, 0',
	X =  227.204  mm,	Y =   -390.088  mm,	Z =   -225.365  mm,
	W =  90.000 deg,	P =   89.765 deg,	R =   30.000 deg
};
P[562]{
   GP1:
	UF : 0, UT : 6,		CONFIG : 'N U T, 0, 0, 0',
	X =  227.444  mm,	Y =   -389.982  mm,	Z =   -224.962  mm,
	W =  90.000 deg,	P =   89.765 deg,	R =   30.000 deg
};
P[563]{
   GP1:
	UF : 0, UT : 6,		CONFIG : 'N U T, 0, 0, 0',
	X =  227.842  mm,	Y =   -389.684  mm,	Z =   -225.808  mm,
	W =  90.000 deg,	P =   89.765 deg,	R =   30.000 deg
};
P[564]{
   GP1:
	UF : 0, UT : 6,		CONFIG : 'N U T, 0, 0, 0',
	X =  228.143  mm,	Y =   -389.577  mm,	Z =   -224.984  mm,
	W =  90.000 deg,	P =   89.765 deg,	R =   30.000 deg
};
P[565]{
   GP1:
	UF : 0, UT : 6,		CONFIG : 'N U T, 0, 0, 0',
	X =  228.461  mm,	Y =   -389.397  mm,	Z =   -224.932  mm,
	W =  90.000 deg,	P =   89.765 deg,	R =   30.000 deg
};
P[566]{
   GP1:
	UF : 0, UT : 6,		CONFIG : 'N U T, 0, 0, 0',
	X =  228.760  mm,	Y =   -389.151  mm,	Z =   -225.837  mm,
	W =  90.000 deg,	P =   89.765 deg,	R =   30.000 deg
};
P[567]{
   GP1:
	UF : 0, UT : 6,		CONFIG : 'N U T, 0, 0, 0',
	X =  228.969  mm,	Y =   -389.072  mm,	Z =   -225.339  mm,
	W =  90.000 deg,	P =   89.765 deg,	R =   30.000 deg
};
P[568]{
   GP1:
	UF : 0, UT : 6,		CONFIG : 'N U T, 0, 0, 0',
	X =  229.080  mm,	Y =   -388.961  mm,	Z =   -225.908  mm,
	W =  90.000 deg,	P =   89.765 deg,	R =   30.000 deg
};
P[569]{
   GP1:
	UF : 0, UT : 6,		CONFIG : 'N U T, 0, 0, 0',
	X =  229.313  mm,	Y =   -388.891  mm,	Z =   -225.105  mm,
	W =  90.000 deg,	P =   89.765 deg,	R =   30.000 deg
};
P[570]{
   GP1:
	UF : 0, UT : 6,		CONFIG : 'N U T, 0, 0, 0',
	X =  229.431  mm,	Y =   -388.802  mm,	Z =   -225.358  mm,
	W =  90.000 deg,	P =   89.765 deg,	R =   30.000 deg
};
P[571]{
   GP1:
	UF : 0, UT : 6,		CONFIG : 'N U T, 0, 0, 0',
	X =  229.961  mm,	Y =   -388.530  mm,	Z =   -224.942  mm,
	W =  90.000 deg,	P =   89.765 deg,	R =   30.000 deg
};
P[572]{
   GP1:
	UF : 0, UT : 6,		CONFIG : 'N U T, 0, 0, 0',
	X =  230.290  mm,	Y =   -388.273  mm,	Z =   -225.777  mm,
	W =  90.000 deg,	P =   89.765 deg,	R =   30.000 deg
};
P[573]{
   GP1:
	UF : 0, UT : 6,		CONFIG : 'N U T, 0, 0, 0',
	X =  230.262  mm,	Y =   -388.357  mm,	Z =   -224.933  mm,
	W =  90.000 deg,	P =   89.765 deg,	R =   30.000 deg
};
P[574]{
   GP1:
	UF : 0, UT : 6,		CONFIG : 'N U T, 0, 0, 0',
	X =  230.551  mm,	Y =   -388.189  mm,	Z =   -224.941  mm,
	W =  90.000 deg,	P =   89.765 deg,	R =   30.000 deg
};
P[575]{
   GP1:
	UF : 0, UT : 6,		CONFIG : 'N U T, 0, 0, 0',
	X =  231.221  mm,	Y =   -387.730  mm,	Z =   -225.842  mm,
	W =  90.000 deg,	P =   89.765 deg,	R =   30.000 deg
};
P[576]{
   GP1:
	UF : 0, UT : 6,		CONFIG : 'N U T, 0, 0, 0',
	X =  231.524  mm,	Y =   -387.596  mm,	Z =   -225.339  mm,
	W =  90.000 deg,	P =   89.765 deg,	R =   30.000 deg
};
P[577]{
   GP1:
	UF : 0, UT : 6,		CONFIG : 'N U T, 0, 0, 0',
	X =  231.779  mm,	Y =   -387.448  mm,	Z =   -225.341  mm,
	W =  90.000 deg,	P =   89.765 deg,	R =   30.000 deg
};
P[578]{
   GP1:
	UF : 0, UT : 6,		CONFIG : 'N U T, 0, 0, 0',
	X =  231.886  mm,	Y =   -387.348  mm,	Z =   -225.817  mm,
	W =  90.000 deg,	P =   89.765 deg,	R =   30.000 deg
};
P[579]{
   GP1:
	UF : 0, UT : 6,		CONFIG : 'N U T, 0, 0, 0',
	X =  232.411  mm,	Y =   -387.115  mm,	Z =   -224.944  mm,
	W =  90.000 deg,	P =   89.765 deg,	R =   30.000 deg
};
P[580]{
   GP1:
	UF : 0, UT : 6,		CONFIG : 'N U T, 0, 0, 0',
	X =  232.704  mm,	Y =   -386.873  mm,	Z =   -225.847  mm,
	W =  90.000 deg,	P =   89.765 deg,	R =   30.000 deg
};
P[581]{
   GP1:
	UF : 0, UT : 6,		CONFIG : 'N U T, 0, 0, 0',
	X =  233.070  mm,	Y =   -386.661  mm,	Z =   -225.857  mm,
	W =  90.000 deg,	P =   89.765 deg,	R =   30.000 deg
};
P[582]{
   GP1:
	UF : 0, UT : 6,		CONFIG : 'N U T, 0, 0, 0',
	X =  233.354  mm,	Y =   -386.571  mm,	Z =   -224.940  mm,
	W =  90.000 deg,	P =   89.765 deg,	R =   30.000 deg
};
P[583]{
   GP1:
	UF : 0, UT : 6,		CONFIG : 'N U T, 0, 0, 0',
	X =  233.702  mm,	Y =   -386.334  mm,	Z =   -225.387  mm,
	W =  90.000 deg,	P =   89.765 deg,	R =   30.000 deg
};
P[584]{
   GP1:
	UF : 0, UT : 6,		CONFIG : 'N U T, 0, 0, 0',
	X =  234.018  mm,	Y =   -386.113  mm,	Z =   -225.871  mm,
	W =  90.000 deg,	P =   89.765 deg,	R =   30.000 deg
};
P[585]{
   GP1:
	UF : 0, UT : 6,		CONFIG : 'N U T, 0, 0, 0',
	X =  234.251  mm,	Y =   -386.052  mm,	Z =   -224.950  mm,
	W =  90.000 deg,	P =   89.765 deg,	R =   30.000 deg
};
P[586]{
   GP1:
	UF : 0, UT : 6,		CONFIG : 'N U T, 0, 0, 0',
	X =  234.584  mm,	Y =   -385.784  mm,	Z =   -225.892  mm,
	W =  90.000 deg,	P =   89.765 deg,	R =   30.000 deg
};
P[587]{
   GP1:
	UF : 0, UT : 6,		CONFIG : 'N U T, 0, 0, 0',
	X =  234.750  mm,	Y =   -385.728  mm,	Z =   -225.408  mm,
	W =  90.000 deg,	P =   89.765 deg,	R =   30.000 deg
};
P[588]{
   GP1:
	UF : 0, UT : 6,		CONFIG : 'N U T, 0, 0, 0',
	X =  235.222  mm,	Y =   -385.416  mm,	Z =   -225.883  mm,
	W =  90.000 deg,	P =   89.765 deg,	R =   30.000 deg
};
P[589]{
   GP1:
	UF : 0, UT : 6,		CONFIG : 'N U T, 0, 0, 0',
	X =  235.479  mm,	Y =   -385.268  mm,	Z =   -225.881  mm,
	W =  90.000 deg,	P =   89.765 deg,	R =   30.000 deg
};
P[590]{
   GP1:
	UF : 0, UT : 6,		CONFIG : 'N U T, 0, 0, 0',
	X =  235.764  mm,	Y =   -385.148  mm,	Z =   -225.328  mm,
	W =  90.000 deg,	P =   89.765 deg,	R =   30.000 deg
};
P[591]{
   GP1:
	UF : 0, UT : 6,		CONFIG : 'N U T, 0, 0, 0',
	X =  235.805  mm,	Y =   -385.077  mm,	Z =   -225.922  mm,
	W =  90.000 deg,	P =   89.765 deg,	R =   30.000 deg
};
P[592]{
   GP1:
	UF : 0, UT : 6,		CONFIG : 'N U T, 0, 0, 0',
	X =  236.079  mm,	Y =   -384.959  mm,	Z =   -225.416  mm,
	W =  90.000 deg,	P =   89.765 deg,	R =   30.000 deg
};
P[593]{
   GP1:
	UF : 0, UT : 6,		CONFIG : 'N U T, 0, 0, 0',
	X =  236.439  mm,	Y =   -384.715  mm,	Z =   -225.869  mm,
	W =  90.000 deg,	P =   89.765 deg,	R =   30.000 deg
};
P[594]{
   GP1:
	UF : 0, UT : 6,		CONFIG : 'N U T, 0, 0, 0',
	X =  236.695  mm,	Y =   -384.606  mm,	Z =   -225.387  mm,
	W =  90.000 deg,	P =   89.765 deg,	R =   30.000 deg
};
P[595]{
   GP1:
	UF : 0, UT : 6,		CONFIG : 'N U T, 0, 0, 0',
	X =  236.741  mm,	Y =   -384.611  mm,	Z =   -225.000  mm,
	W =  90.000 deg,	P =   89.765 deg,	R =   30.000 deg
};
P[596]{
   GP1:
	UF : 0, UT : 6,		CONFIG : 'N U T, 0, 0, 0',
	X =  237.093  mm,	Y =   -384.411  mm,	Z =   -224.955  mm,
	W =  90.000 deg,	P =   89.765 deg,	R =   30.000 deg
};
P[597]{
   GP1:
	UF : 0, UT : 6,		CONFIG : 'N U T, 0, 0, 0',
	X =  237.353  mm,	Y =   -384.259  mm,	Z =   -224.978  mm,
	W =  90.000 deg,	P =   89.765 deg,	R =   30.000 deg
};
P[598]{
   GP1:
	UF : 0, UT : 6,		CONFIG : 'N U T, 0, 0, 0',
	X =  237.648  mm,	Y =   -384.054  mm,	Z =   -225.411  mm,
	W =  90.000 deg,	P =   89.765 deg,	R =   30.000 deg
};
P[599]{
   GP1:
	UF : 0, UT : 6,		CONFIG : 'N U T, 0, 0, 0',
	X =  237.669  mm,	Y =   -384.009  mm,	Z =   -225.820  mm,
	W =  90.000 deg,	P =   89.765 deg,	R =   30.000 deg
};
P[600]{
   GP1:
	UF : 0, UT : 6,		CONFIG : 'N U T, 0, 0, 0',
	X =  237.972  mm,	Y =   -383.831  mm,	Z =   -225.856  mm,
	W =  90.000 deg,	P =   89.765 deg,	R =   30.000 deg
};
P[601]{
   GP1:
	UF : 0, UT : 6,		CONFIG : 'N U T, 0, 0, 0',
	X =  238.234  mm,	Y =   -383.720  mm,	Z =   -225.344  mm,
	W =  90.000 deg,	P =   89.765 deg,	R =   30.000 deg
};
P[602]{
   GP1:
	UF : 0, UT : 6,		CONFIG : 'N U T, 0, 0, 0',
	X =  238.600  mm,	Y =   -383.464  mm,	Z =   -225.913  mm,
	W =  90.000 deg,	P =   89.765 deg,	R =   30.000 deg
};
P[603]{
   GP1:
	UF : 0, UT : 6,		CONFIG : 'N U T, 0, 0, 0',
	X =  238.858  mm,	Y =   -383.337  mm,	Z =   -225.637  mm,
	W =  90.000 deg,	P =   89.765 deg,	R =   30.000 deg
};
P[604]{
   GP1:
	UF : 0, UT : 6,		CONFIG : 'N U T, 0, 0, 0',
	X =  239.286  mm,	Y =   -383.111  mm,	Z =   -225.378  mm,
	W =  90.000 deg,	P =   89.765 deg,	R =   30.000 deg
};
P[605]{
   GP1:
	UF : 0, UT : 6,		CONFIG : 'N U T, 0, 0, 0',
	X =  239.396  mm,	Y =   -383.048  mm,	Z =   -225.375  mm,
	W =  90.000 deg,	P =   89.765 deg,	R =   30.000 deg
};
P[606]{
   GP1:
	UF : 0, UT : 6,		CONFIG : 'N U T, 0, 0, 0',
	X =  239.483  mm,	Y =   -383.023  mm,	Z =   -225.059  mm,
	W =  90.000 deg,	P =   89.765 deg,	R =   30.000 deg
};
P[607]{
   GP1:
	UF : 0, UT : 6,		CONFIG : 'N U T, 0, 0, 0',
	X =  239.820  mm,	Y =   -382.762  mm,	Z =   -225.882  mm,
	W =  90.000 deg,	P =   89.765 deg,	R =   30.000 deg
};
P[608]{
   GP1:
	UF : 0, UT : 6,		CONFIG : 'N U T, 0, 0, 0',
	X =  240.385  mm,	Y =   -382.440  mm,	Z =   -225.833  mm,
	W =  90.000 deg,	P =   89.765 deg,	R =   30.000 deg
};
P[609]{
   GP1:
	UF : 0, UT : 6,		CONFIG : 'N U T, 0, 0, 0',
	X =  240.466  mm,	Y =   -382.464  mm,	Z =   -224.948  mm,
	W =  90.000 deg,	P =   89.765 deg,	R =   30.000 deg
};
P[610]{
   GP1:
	UF : 0, UT : 6,		CONFIG : 'N U T, 0, 0, 0',
	X =  240.667  mm,	Y =   -382.310  mm,	Z =   -225.415  mm,
	W =  90.000 deg,	P =   89.765 deg,	R =   30.000 deg
};
P[611]{
   GP1:
	UF : 0, UT : 6,		CONFIG : 'N U T, 0, 0, 0',
	X =  241.011  mm,	Y =   -382.080  mm,	Z =   -225.816  mm,
	W =  90.000 deg,	P =   89.765 deg,	R =   30.000 deg
};
P[612]{
   GP1:
	UF : 0, UT : 6,		CONFIG : 'N U T, 0, 0, 0',
	X =  241.057  mm,	Y =   -382.114  mm,	Z =   -225.054  mm,
	W =  90.000 deg,	P =   89.765 deg,	R =   30.000 deg
};
P[613]{
   GP1:
	UF : 0, UT : 6,		CONFIG : 'N U T, 0, 0, 0',
	X =  241.651  mm,	Y =   -381.705  mm,	Z =   -225.880  mm,
	W =  90.000 deg,	P =   89.765 deg,	R =   30.000 deg
};
P[614]{
   GP1:
	UF : 0, UT : 6,		CONFIG : 'N U T, 0, 0, 0',
	X =  241.657  mm,	Y =   -381.744  mm,	Z =   -225.353  mm,
	W =  90.000 deg,	P =   89.765 deg,	R =   30.000 deg
};
P[615]{
   GP1:
	UF : 0, UT : 6,		CONFIG : 'N U T, 0, 0, 0',
	X =  241.682  mm,	Y =   -381.762  mm,	Z =   -224.954  mm,
	W =  90.000 deg,	P =   89.765 deg,	R =   30.000 deg
};
P[616]{
   GP1:
	UF : 0, UT : 6,		CONFIG : 'N U T, 0, 0, 0',
	X =  241.916  mm,	Y =   -381.590  mm,	Z =   -225.405  mm,
	W =  90.000 deg,	P =   89.765 deg,	R =   30.000 deg
};
P[617]{
   GP1:
	UF : 0, UT : 6,		CONFIG : 'N U T, 0, 0, 0',
	X =  242.020  mm,	Y =   -381.568  mm,	Z =   -224.939  mm,
	W =  90.000 deg,	P =   89.765 deg,	R =   30.000 deg
};
P[618]{
   GP1:
	UF : 0, UT : 6,		CONFIG : 'N U T, 0, 0, 0',
	X =  242.136  mm,	Y =   -381.466  mm,	Z =   -225.368  mm,
	W =  90.000 deg,	P =   89.765 deg,	R =   30.000 deg
};
P[619]{
   GP1:
	UF : 0, UT : 6,		CONFIG : 'N U T, 0, 0, 0',
	X =  242.299  mm,	Y =   -381.335  mm,	Z =   -225.829  mm,
	W =  90.000 deg,	P =   89.765 deg,	R =   30.000 deg
};
P[620]{
   GP1:
	UF : 0, UT : 6,		CONFIG : 'N U T, 0, 0, 0',
	X =  242.862  mm,	Y =   -381.010  mm,	Z =   -225.826  mm,
	W =  90.000 deg,	P =   89.765 deg,	R =   30.000 deg
};
P[621]{
   GP1:
	UF : 0, UT : 6,		CONFIG : 'N U T, 0, 0, 0',
	X =  242.967  mm,	Y =   -380.988  mm,	Z =   -225.344  mm,
	W =  90.000 deg,	P =   89.765 deg,	R =   30.000 deg
};
P[622]{
   GP1:
	UF : 0, UT : 6,		CONFIG : 'N U T, 0, 0, 0',
	X =  243.191  mm,	Y =   -380.884  mm,	Z =   -225.033  mm,
	W =  90.000 deg,	P =   89.765 deg,	R =   30.000 deg
};
P[623]{
   GP1:
	UF : 0, UT : 6,		CONFIG : 'N U T, 0, 0, 0',
	X =  243.329  mm,	Y =   -380.773  mm,	Z =   -225.413  mm,
	W =  90.000 deg,	P =   89.765 deg,	R =   30.000 deg
};
P[624]{
   GP1:
	UF : 0, UT : 6,		CONFIG : 'N U T, 0, 0, 0',
	X =  243.446  mm,	Y =   -380.710  mm,	Z =   -225.365  mm,
	W =  90.000 deg,	P =   89.765 deg,	R =   30.000 deg
};
P[625]{
   GP1:
	UF : 0, UT : 6,		CONFIG : 'N U T, 0, 0, 0',
	X =  243.789  mm,	Y =   -380.472  mm,	Z =   -225.855  mm,
	W =  90.000 deg,	P =   89.765 deg,	R =   30.000 deg
};
P[626]{
   GP1:
	UF : 0, UT : 6,		CONFIG : 'N U T, 0, 0, 0',
	X =  243.833  mm,	Y =   -380.489  mm,	Z =   -225.337  mm,
	W =  90.000 deg,	P =   89.765 deg,	R =   30.000 deg
};
P[627]{
   GP1:
	UF : 0, UT : 6,		CONFIG : 'N U T, 0, 0, 0',
	X =  243.997  mm,	Y =   -380.389  mm,	Z =   -225.404  mm,
	W =  90.000 deg,	P =   89.765 deg,	R =   30.000 deg
};
P[628]{
   GP1:
	UF : 0, UT : 6,		CONFIG : 'N U T, 0, 0, 0',
	X =  244.143  mm,	Y =   -380.341  mm,	Z =   -224.949  mm,
	W =  90.000 deg,	P =   89.765 deg,	R =   30.000 deg
};
P[629]{
   GP1:
	UF : 0, UT : 6,		CONFIG : 'N U T, 0, 0, 0',
	X =  244.128  mm,	Y =   -380.271  mm,	Z =   -225.924  mm,
	W =  90.000 deg,	P =   89.765 deg,	R =   30.000 deg
};
P[630]{
   GP1:
	UF : 0, UT : 6,		CONFIG : 'N U T, 0, 0, 0',
	X =  244.422  mm,	Y =   -380.111  mm,	Z =   -225.802  mm,
	W =  90.000 deg,	P =   89.765 deg,	R =   30.000 deg
};
P[631]{
   GP1:
	UF : 0, UT : 6,		CONFIG : 'N U T, 0, 0, 0',
	X =  244.455  mm,	Y =   -380.163  mm,	Z =   -224.926  mm,
	W =  90.000 deg,	P =   89.765 deg,	R =   30.000 deg
};
P[632]{
   GP1:
	UF : 0, UT : 6,		CONFIG : 'N U T, 0, 0, 0',
	X =  244.451  mm,	Y =   -380.132  mm,	Z =   -225.328  mm,
	W =  90.000 deg,	P =   89.765 deg,	R =   30.000 deg
};
P[633]{
   GP1:
	UF : 0, UT : 6,		CONFIG : 'N U T, 0, 0, 0',
	X =  245.272  mm,	Y =   -379.659  mm,	Z =   -225.320  mm,
	W =  90.000 deg,	P =   89.765 deg,	R =   30.000 deg
};
P[634]{
   GP1:
	UF : 0, UT : 6,		CONFIG : 'N U T, 0, 0, 0',
	X =  245.523  mm,	Y =   -379.514  mm,	Z =   -225.322  mm,
	W =  90.000 deg,	P =   89.765 deg,	R =   30.000 deg
};
P[635]{
   GP1:
	UF : 0, UT : 6,		CONFIG : 'N U T, 0, 0, 0',
	X =  245.626  mm,	Y =   -379.406  mm,	Z =   -225.922  mm,
	W =  90.000 deg,	P =   89.765 deg,	R =   30.000 deg
};
P[636]{
   GP1:
	UF : 0, UT : 6,		CONFIG : 'N U T, 0, 0, 0',
	X =  245.945  mm,	Y =   -379.226  mm,	Z =   -225.871  mm,
	W =  90.000 deg,	P =   89.765 deg,	R =   30.000 deg
};
P[637]{
   GP1:
	UF : 0, UT : 6,		CONFIG : 'N U T, 0, 0, 0',
	X =  246.321  mm,	Y =   -379.048  mm,	Z =   -225.388  mm,
	W =  90.000 deg,	P =   89.765 deg,	R =   30.000 deg
};
P[638]{
   GP1:
	UF : 0, UT : 6,		CONFIG : 'N U T, 0, 0, 0',
	X =  246.436  mm,	Y =   -378.982  mm,	Z =   -225.386  mm,
	W =  90.000 deg,	P =   89.765 deg,	R =   30.000 deg
};
P[639]{
   GP1:
	UF : 0, UT : 6,		CONFIG : 'N U T, 0, 0, 0',
	X =  246.616  mm,	Y =   -378.914  mm,	Z =   -224.933  mm,
	W =  90.000 deg,	P =   89.765 deg,	R =   30.000 deg
};
P[640]{
   GP1:
	UF : 0, UT : 6,		CONFIG : 'N U T, 0, 0, 0',
	X =  246.813  mm,	Y =   -378.762  mm,	Z =   -225.399  mm,
	W =  90.000 deg,	P =   89.765 deg,	R =   30.000 deg
};
P[641]{
   GP1:
	UF : 0, UT : 6,		CONFIG : 'N U T, 0, 0, 0',
	X =  247.228  mm,	Y =   -378.561  mm,	Z =   -224.929  mm,
	W =  90.000 deg,	P =   89.765 deg,	R =   30.000 deg
};
P[642]{
   GP1:
	UF : 0, UT : 6,		CONFIG : 'N U T, 0, 0, 0',
	X =  247.322  mm,	Y =   -378.470  mm,	Z =   -225.390  mm,
	W =  90.000 deg,	P =   89.765 deg,	R =   30.000 deg
};
P[643]{
   GP1:
	UF : 0, UT : 6,		CONFIG : 'N U T, 0, 0, 0',
	X =  247.499  mm,	Y =   -378.335  mm,	Z =   -225.793  mm,
	W =  90.000 deg,	P =   89.765 deg,	R =   30.000 deg
};
P[644]{
   GP1:
	UF : 0, UT : 6,		CONFIG : 'N U T, 0, 0, 0',
	X =  247.760  mm,	Y =   -378.218  mm,	Z =   -225.374  mm,
	W =  90.000 deg,	P =   89.765 deg,	R =   30.000 deg
};
P[645]{
   GP1:
	UF : 0, UT : 6,		CONFIG : 'N U T, 0, 0, 0',
	X =  248.085  mm,	Y =   -377.995  mm,	Z =   -225.818  mm,
	W =  90.000 deg,	P =   89.765 deg,	R =   30.000 deg
};
P[646]{
   GP1:
	UF : 0, UT : 6,		CONFIG : 'N U T, 0, 0, 0',
	X =  248.384  mm,	Y =   -377.816  mm,	Z =   -225.894  mm,
	W =  90.000 deg,	P =   89.765 deg,	R =   30.000 deg
};
P[647]{
   GP1:
	UF : 0, UT : 6,		CONFIG : 'N U T, 0, 0, 0',
	X =  248.435  mm,	Y =   -377.829  mm,	Z =   -225.369  mm,
	W =  90.000 deg,	P =   89.765 deg,	R =   30.000 deg
};
P[648]{
   GP1:
	UF : 0, UT : 6,		CONFIG : 'N U T, 0, 0, 0',
	X =  248.720  mm,	Y =   -377.698  mm,	Z =   -224.950  mm,
	W =  90.000 deg,	P =   89.765 deg,	R =   30.000 deg
};
P[649]{
   GP1:
	UF : 0, UT : 6,		CONFIG : 'N U T, 0, 0, 0',
	X =  248.727  mm,	Y =   -377.624  mm,	Z =   -225.823  mm,
	W =  90.000 deg,	P =   89.765 deg,	R =   30.000 deg
};
P[650]{
   GP1:
	UF : 0, UT : 6,		CONFIG : 'N U T, 0, 0, 0',
	X =  249.026  mm,	Y =   -377.491  mm,	Z =   -225.335  mm,
	W =  90.000 deg,	P =   89.765 deg,	R =   30.000 deg
};
P[651]{
   GP1:
	UF : 0, UT : 6,		CONFIG : 'N U T, 0, 0, 0',
	X =  249.355  mm,	Y =   -377.320  mm,	Z =   -225.096  mm,
	W =  90.000 deg,	P =   89.765 deg,	R =   30.000 deg
};
P[652]{
   GP1:
	UF : 0, UT : 6,		CONFIG : 'N U T, 0, 0, 0',
	X =  249.339  mm,	Y =   -377.274  mm,	Z =   -225.774  mm,
	W =  90.000 deg,	P =   89.765 deg,	R =   30.000 deg
};
P[653]{
   GP1:
	UF : 0, UT : 6,		CONFIG : 'N U T, 0, 0, 0',
	X =  249.677  mm,	Y =   -377.068  mm,	Z =   -225.918  mm,
	W =  90.000 deg,	P =   89.765 deg,	R =   30.000 deg
};
P[654]{
   GP1:
	UF : 0, UT : 6,		CONFIG : 'N U T, 0, 0, 0',
	X =  249.867  mm,	Y =   -376.998  mm,	Z =   -225.416  mm,
	W =  90.000 deg,	P =   89.765 deg,	R =   30.000 deg
};
P[655]{
   GP1:
	UF : 0, UT : 6,		CONFIG : 'N U T, 0, 0, 0',
	X =  250.198  mm,	Y =   -376.775  mm,	Z =   -225.823  mm,
	W =  90.000 deg,	P =   89.765 deg,	R =   30.000 deg
};
P[656]{
   GP1:
	UF : 0, UT : 6,		CONFIG : 'N U T, 0, 0, 0',
	X =  250.359  mm,	Y =   -376.750  mm,	Z =   -224.979  mm,
	W =  90.000 deg,	P =   89.765 deg,	R =   30.000 deg
};
P[657]{
   GP1:
	UF : 0, UT : 6,		CONFIG : 'N U T, 0, 0, 0',
	X =  250.512  mm,	Y =   -376.587  mm,	Z =   -225.904  mm,
	W =  90.000 deg,	P =   89.765 deg,	R =   30.000 deg
};
P[658]{
   GP1:
	UF : 0, UT : 6,		CONFIG : 'N U T, 0, 0, 0',
	X =  250.662  mm,	Y =   -376.546  mm,	Z =   -225.329  mm,
	W =  90.000 deg,	P =   89.765 deg,	R =   30.000 deg
};
P[659]{
   GP1:
	UF : 0, UT : 6,		CONFIG : 'N U T, 0, 0, 0',
	X =  250.870  mm,	Y =   -376.383  mm,	Z =   -225.871  mm,
	W =  90.000 deg,	P =   89.765 deg,	R =   30.000 deg
};
P[660]{
   GP1:
	UF : 0, UT : 6,		CONFIG : 'N U T, 0, 0, 0',
	X =  251.161  mm,	Y =   -376.220  mm,	Z =   -225.811  mm,
	W =  90.000 deg,	P =   89.765 deg,	R =   30.000 deg
};
P[661]{
   GP1:
	UF : 0, UT : 6,		CONFIG : 'N U T, 0, 0, 0',
	X =  251.431  mm,	Y =   -376.071  mm,	Z =   -225.717  mm,
	W =  90.000 deg,	P =   89.765 deg,	R =   30.000 deg
};
P[662]{
   GP1:
	UF : 0, UT : 6,		CONFIG : 'N U T, 0, 0, 0',
	X =  251.510  mm,	Y =   -376.086  mm,	Z =   -224.963  mm,
	W =  90.000 deg,	P =   89.765 deg,	R =   30.000 deg
};
P[663]{
   GP1:
	UF : 0, UT : 6,		CONFIG : 'N U T, 0, 0, 0',
	X =  251.835  mm,	Y =   -375.866  mm,	Z =   -225.367  mm,
	W =  90.000 deg,	P =   89.765 deg,	R =   30.000 deg
};
P[664]{
   GP1:
	UF : 0, UT : 6,		CONFIG : 'N U T, 0, 0, 0',
	X =  252.144  mm,	Y =   -375.724  mm,	Z =   -224.927  mm,
	W =  90.000 deg,	P =   89.765 deg,	R =   30.000 deg
};
P[665]{
   GP1:
	UF : 0, UT : 6,		CONFIG : 'N U T, 0, 0, 0',
	X =  252.539  mm,	Y =   -375.459  mm,	Z =   -225.370  mm,
	W =  90.000 deg,	P =   89.765 deg,	R =   30.000 deg
};
P[666]{
   GP1:
	UF : 0, UT : 6,		CONFIG : 'N U T, 0, 0, 0',
	X =  252.711  mm,	Y =   -375.322  mm,	Z =   -225.842  mm,
	W =  90.000 deg,	P =   89.765 deg,	R =   30.000 deg
};
P[667]{
   GP1:
	UF : 0, UT : 6,		CONFIG : 'N U T, 0, 0, 0',
	X =  252.790  mm,	Y =   -375.348  mm,	Z =   -224.952  mm,
	W =  90.000 deg,	P =   89.765 deg,	R =   30.000 deg
};
P[668]{
   GP1:
	UF : 0, UT : 6,		CONFIG : 'N U T, 0, 0, 0',
	X =  252.956  mm,	Y =   -375.174  mm,	Z =   -225.925  mm,
	W =  90.000 deg,	P =   89.765 deg,	R =   30.000 deg
};
P[669]{
   GP1:
	UF : 0, UT : 6,		CONFIG : 'N U T, 0, 0, 0',
	X =  253.157  mm,	Y =   -375.102  mm,	Z =   -225.380  mm,
	W =  90.000 deg,	P =   89.765 deg,	R =   30.000 deg
};
P[670]{
   GP1:
	UF : 0, UT : 6,		CONFIG : 'N U T, 0, 0, 0',
	X =  253.518  mm,	Y =   -374.896  mm,	Z =   -225.344  mm,
	W =  90.000 deg,	P =   89.765 deg,	R =   30.000 deg
};
P[671]{
   GP1:
	UF : 0, UT : 6,		CONFIG : 'N U T, 0, 0, 0',
	X =  253.647  mm,	Y =   -374.782  mm,	Z =   -225.836  mm,
	W =  90.000 deg,	P =   89.765 deg,	R =   30.000 deg
};
P[672]{
   GP1:
	UF : 0, UT : 6,		CONFIG : 'N U T, 0, 0, 0',
	X =  253.928  mm,	Y =   -374.617  mm,	Z =   -225.872  mm,
	W =  90.000 deg,	P =   89.765 deg,	R =   30.000 deg
};
P[673]{
   GP1:
	UF : 0, UT : 6,		CONFIG : 'N U T, 0, 0, 0',
	X =  254.618  mm,	Y =   -374.291  mm,	Z =   -224.970  mm,
	W =  90.000 deg,	P =   89.765 deg,	R =   30.000 deg
};
P[674]{
   GP1:
	UF : 0, UT : 6,		CONFIG : 'N U T, 0, 0, 0',
	X =  254.548  mm,	Y =   -374.258  mm,	Z =   -225.877  mm,
	W =  90.000 deg,	P =   89.765 deg,	R =   30.000 deg
};
P[675]{
   GP1:
	UF : 0, UT : 6,		CONFIG : 'N U T, 0, 0, 0',
	X =  254.833  mm,	Y =   -374.101  mm,	Z =   -225.784  mm,
	W =  90.000 deg,	P =   89.765 deg,	R =   30.000 deg
};
P[676]{
   GP1:
	UF : 0, UT : 6,		CONFIG : 'N U T, 0, 0, 0',
	X =  254.916  mm,	Y =   -374.117  mm,	Z =   -225.006  mm,
	W =  90.000 deg,	P =   89.765 deg,	R =   30.000 deg
};
P[677]{
   GP1:
	UF : 0, UT : 6,		CONFIG : 'N U T, 0, 0, 0',
	X =  255.082  mm,	Y =   -373.949  mm,	Z =   -225.895  mm,
	W =  90.000 deg,	P =   89.765 deg,	R =   30.000 deg
};
P[678]{
   GP1:
	UF : 0, UT : 6,		CONFIG : 'N U T, 0, 0, 0',
	X =  255.212  mm,	Y =   -373.949  mm,	Z =   -224.954  mm,
	W =  90.000 deg,	P =   89.765 deg,	R =   30.000 deg
};
P[679]{
   GP1:
	UF : 0, UT : 6,		CONFIG : 'N U T, 0, 0, 0',
	X =  255.782  mm,	Y =   -373.545  mm,	Z =   -225.881  mm,
	W =  90.000 deg,	P =   89.765 deg,	R =   30.000 deg
};
P[680]{
   GP1:
	UF : 0, UT : 6,		CONFIG : 'N U T, 0, 0, 0',
	X =  255.863  mm,	Y =   -373.538  mm,	Z =   -225.385  mm,
	W =  90.000 deg,	P =   89.765 deg,	R =   30.000 deg
};
P[681]{
   GP1:
	UF : 0, UT : 6,		CONFIG : 'N U T, 0, 0, 0',
	X =  256.059  mm,	Y =   -373.389  mm,	Z =   -225.836  mm,
	W =  90.000 deg,	P =   89.765 deg,	R =   30.000 deg
};
P[682]{
   GP1:
	UF : 0, UT : 6,		CONFIG : 'N U T, 0, 0, 0',
	X =  256.360  mm,	Y =   -373.216  mm,	Z =   -225.825  mm,
	W =  90.000 deg,	P =   89.765 deg,	R =   30.000 deg
};
P[683]{
   GP1:
	UF : 0, UT : 6,		CONFIG : 'N U T, 0, 0, 0',
	X =  256.646  mm,	Y =   -373.087  mm,	Z =   -225.373  mm,
	W =  90.000 deg,	P =   89.765 deg,	R =   30.000 deg
};
P[684]{
   GP1:
	UF : 0, UT : 6,		CONFIG : 'N U T, 0, 0, 0',
	X =  256.948  mm,	Y =   -372.876  mm,	Z =   -225.832  mm,
	W =  90.000 deg,	P =   89.765 deg,	R =   30.000 deg
};
P[685]{
   GP1:
	UF : 0, UT : 6,		CONFIG : 'N U T, 0, 0, 0',
	X =  257.292  mm,	Y =   -372.671  mm,	Z =   -225.911  mm,
	W =  90.000 deg,	P =   89.765 deg,	R =   30.000 deg
};
P[686]{
   GP1:
	UF : 0, UT : 6,		CONFIG : 'N U T, 0, 0, 0',
	X =  257.580  mm,	Y =   -372.508  mm,	Z =   -225.875  mm,
	W =  90.000 deg,	P =   89.765 deg,	R =   30.000 deg
};
P[687]{
   GP1:
	UF : 0, UT : 6,		CONFIG : 'N U T, 0, 0, 0',
	X =  257.861  mm,	Y =   -372.347  mm,	Z =   -225.855  mm,
	W =  90.000 deg,	P =   89.765 deg,	R =   30.000 deg
};
P[688]{
   GP1:
	UF : 0, UT : 6,		CONFIG : 'N U T, 0, 0, 0',
	X =  258.196  mm,	Y =   -372.156  mm,	Z =   -225.826  mm,
	W =  90.000 deg,	P =   89.765 deg,	R =   30.000 deg
};
P[689]{
   GP1:
	UF : 0, UT : 6,		CONFIG : 'N U T, 0, 0, 0',
	X =  258.609  mm,	Y =   -371.982  mm,	Z =   -225.024  mm,
	W =  90.000 deg,	P =   89.765 deg,	R =   30.000 deg
};
P[690]{
   GP1:
	UF : 0, UT : 6,		CONFIG : 'N U T, 0, 0, 0',
	X =  258.806  mm,	Y =   -371.808  mm,	Z =   -225.779  mm,
	W =  90.000 deg,	P =   89.765 deg,	R =   30.000 deg
};
P[691]{
   GP1:
	UF : 0, UT : 6,		CONFIG : 'N U T, 0, 0, 0',
	X =  258.952  mm,	Y =   -371.791  mm,	Z =   -224.939  mm,
	W =  90.000 deg,	P =   89.765 deg,	R =   30.000 deg
};
P[692]{
   GP1:
	UF : 0, UT : 6,		CONFIG : 'N U T, 0, 0, 0',
	X =  259.383  mm,	Y =   -371.465  mm,	Z =   -225.892  mm,
	W =  90.000 deg,	P =   89.765 deg,	R =   30.000 deg
};
P[693]{
   GP1:
	UF : 0, UT : 6,		CONFIG : 'N U T, 0, 0, 0',
	X =  259.469  mm,	Y =   -371.460  mm,	Z =   -225.342  mm,
	W =  90.000 deg,	P =   89.765 deg,	R =   30.000 deg
};
P[694]{
   GP1:
	UF : 0, UT : 6,		CONFIG : 'N U T, 0, 0, 0',
	X =  260.230  mm,	Y =   -371.016  mm,	Z =   -225.405  mm,
	W =  90.000 deg,	P =   89.765 deg,	R =   30.000 deg
};
P[695]{
   GP1:
	UF : 0, UT : 6,		CONFIG : 'N U T, 0, 0, 0',
	X =  260.543  mm,	Y =   -370.834  mm,	Z =   -225.415  mm,
	W =  90.000 deg,	P =   89.765 deg,	R =   30.000 deg
};
P[696]{
   GP1:
	UF : 0, UT : 6,		CONFIG : 'N U T, 0, 0, 0',
	X =  260.754  mm,	Y =   -370.719  mm,	Z =   -225.329  mm,
	W =  90.000 deg,	P =   89.765 deg,	R =   30.000 deg
};
P[697]{
   GP1:
	UF : 0, UT : 6,		CONFIG : 'N U T, 0, 0, 0',
	X =  261.051  mm,	Y =   -370.577  mm,	Z =   -224.965  mm,
	W =  90.000 deg,	P =   89.765 deg,	R =   30.000 deg
};
P[698]{
   GP1:
	UF : 0, UT : 6,		CONFIG : 'N U T, 0, 0, 0',
	X =  261.265  mm,	Y =   -370.381  mm,	Z =   -225.867  mm,
	W =  90.000 deg,	P =   89.765 deg,	R =   30.000 deg
};
P[699]{
   GP1:
	UF : 0, UT : 6,		CONFIG : 'N U T, 0, 0, 0',
	X =  261.708  mm,	Y =   -370.199  mm,	Z =   -224.954  mm,
	W =  90.000 deg,	P =   89.765 deg,	R =   30.000 deg
};
P[700]{
   GP1:
	UF : 0, UT : 6,		CONFIG : 'N U T, 0, 0, 0',
	X =  261.608  mm,	Y =   -370.187  mm,	Z =   -225.816  mm,
	W =  90.000 deg,	P =   89.765 deg,	R =   30.000 deg
};
P[701]{
   GP1:
	UF : 0, UT : 6,		CONFIG : 'N U T, 0, 0, 0',
	X =  261.992  mm,	Y =   -370.036  mm,	Z =   -224.936  mm,
	W =  90.000 deg,	P =   89.765 deg,	R =   30.000 deg
};
P[702]{
   GP1:
	UF : 0, UT : 6,		CONFIG : 'N U T, 0, 0, 0',
	X =  261.887  mm,	Y =   -370.021  mm,	Z =   -225.874  mm,
	W =  90.000 deg,	P =   89.765 deg,	R =   30.000 deg
};
P[703]{
   GP1:
	UF : 0, UT : 6,		CONFIG : 'N U T, 0, 0, 0',
	X =  261.957  mm,	Y =   -370.021  mm,	Z =   -225.372  mm,
	W =  90.000 deg,	P =   89.765 deg,	R =   30.000 deg
};
P[704]{
   GP1:
	UF : 0, UT : 6,		CONFIG : 'N U T, 0, 0, 0',
	X =  262.562  mm,	Y =   -369.706  mm,	Z =   -224.952  mm,
	W =  90.000 deg,	P =   89.765 deg,	R =   30.000 deg
};
P[705]{
   GP1:
	UF : 0, UT : 6,		CONFIG : 'N U T, 0, 0, 0',
	X =  262.651  mm,	Y =   -369.621  mm,	Z =   -225.357  mm,
	W =  90.000 deg,	P =   89.765 deg,	R =   30.000 deg
};
P[706]{
   GP1:
	UF : 0, UT : 6,		CONFIG : 'N U T, 0, 0, 0',
	X =  262.831  mm,	Y =   -369.521  mm,	Z =   -225.316  mm,
	W =  90.000 deg,	P =   89.765 deg,	R =   30.000 deg
};
P[707]{
   GP1:
	UF : 0, UT : 6,		CONFIG : 'N U T, 0, 0, 0',
	X =  262.835  mm,	Y =   -369.473  mm,	Z =   -225.883  mm,
	W =  90.000 deg,	P =   89.765 deg,	R =   30.000 deg
};
P[708]{
   GP1:
	UF : 0, UT : 6,		CONFIG : 'N U T, 0, 0, 0',
	X =  263.208  mm,	Y =   -369.299  mm,	Z =   -225.372  mm,
	W =  90.000 deg,	P =   89.765 deg,	R =   30.000 deg
};
P[709]{
   GP1:
	UF : 0, UT : 6,		CONFIG : 'N U T, 0, 0, 0',
	X =  263.405  mm,	Y =   -369.148  mm,	Z =   -225.827  mm,
	W =  90.000 deg,	P =   89.765 deg,	R =   30.000 deg
};
P[710]{
   GP1:
	UF : 0, UT : 6,		CONFIG : 'N U T, 0, 0, 0',
	X =  263.510  mm,	Y =   -369.129  mm,	Z =   -225.317  mm,
	W =  90.000 deg,	P =   89.765 deg,	R =   30.000 deg
};
P[711]{
   GP1:
	UF : 0, UT : 6,		CONFIG : 'N U T, 0, 0, 0',
	X =  263.762  mm,	Y =   -368.977  mm,	Z =   -225.384  mm,
	W =  90.000 deg,	P =   89.765 deg,	R =   30.000 deg
};
P[712]{
   GP1:
	UF : 0, UT : 6,		CONFIG : 'N U T, 0, 0, 0',
	X =  264.099  mm,	Y =   -368.820  mm,	Z =   -224.929  mm,
	W =  90.000 deg,	P =   89.765 deg,	R =   30.000 deg
};
P[713]{
   GP1:
	UF : 0, UT : 6,		CONFIG : 'N U T, 0, 0, 0',
	X =  264.374  mm,	Y =   -368.623  mm,	Z =   -225.404  mm,
	W =  90.000 deg,	P =   89.765 deg,	R =   30.000 deg
};
P[714]{
   GP1:
	UF : 0, UT : 6,		CONFIG : 'N U T, 0, 0, 0',
	X =  264.738  mm,	Y =   -368.449  mm,	Z =   -224.967  mm,
	W =  90.000 deg,	P =   89.765 deg,	R =   30.000 deg
};
P[715]{
   GP1:
	UF : 0, UT : 6,		CONFIG : 'N U T, 0, 0, 0',
	X =  265.046  mm,	Y =   -368.215  mm,	Z =   -224.961  mm,
	W =  90.000 deg,	P =   89.765 deg,	R =   30.000 deg
};
P[716]{
   GP1:
	UF : 0, UT : 6,		CONFIG : 'N U T, 0, 0, 0',
	X =  264.922  mm,	Y =   -368.223  mm,	Z =   -225.798  mm,
	W =  90.000 deg,	P =   89.765 deg,	R =   30.000 deg
};
P[717]{
   GP1:
	UF : 0, UT : 6,		CONFIG : 'N U T, 0, 0, 0',
	X =  265.043  mm,	Y =   -368.011  mm,	Z =   -225.859  mm,
	W =  90.000 deg,	P =   89.765 deg,	R =   30.000 deg
};
P[718]{
   GP1:
	UF : 0, UT : 6,		CONFIG : 'N U T, 0, 0, 0',
	X =  265.129  mm,	Y =   -367.854  mm,	Z =   -224.929  mm,
	W =  90.000 deg,	P =   89.765 deg,	R =   30.000 deg
};
P[719]{
   GP1:
	UF : 0, UT : 6,		CONFIG : 'N U T, 0, 0, 0',
	X =  264.965  mm,	Y =   -367.806  mm,	Z =   -225.878  mm,
	W =  90.000 deg,	P =   89.765 deg,	R =   30.000 deg
};
P[720]{
   GP1:
	UF : 0, UT : 6,		CONFIG : 'N U T, 0, 0, 0',
	X =  264.906  mm,	Y =   -367.646  mm,	Z =   -224.950  mm,
	W =  90.000 deg,	P =   89.765 deg,	R =   30.000 deg
};
P[721]{
   GP1:
	UF : 0, UT : 6,		CONFIG : 'N U T, 0, 0, 0',
	X =  264.703  mm,	Y =   -367.604  mm,	Z =   -225.881  mm,
	W =  90.000 deg,	P =   89.765 deg,	R =   30.000 deg
};
P[722]{
   GP1:
	UF : 0, UT : 6,		CONFIG : 'N U T, 0, 0, 0',
	X =  264.534  mm,	Y =   -367.499  mm,	Z =   -225.835  mm,
	W =  90.000 deg,	P =   89.765 deg,	R =   30.000 deg
};
P[723]{
   GP1:
	UF : 0, UT : 6,		CONFIG : 'N U T, 0, 0, 0',
	X =  264.133  mm,	Y =   -367.358  mm,	Z =   -225.818  mm,
	W =  90.000 deg,	P =   89.765 deg,	R =   30.000 deg
};
P[724]{
   GP1:
	UF : 0, UT : 6,		CONFIG : 'N U T, 0, 0, 0',
	X =  293.100  mm,	Y =   -362.853  mm,	Z =   -224.936  mm,
	W =  0.235 deg,	P =   0.000 deg,	R =   30.000 deg
};
P[725]{
   GP1:
	UF : 0, UT : 6,		CONFIG : 'N U T, 0, 0, 0',
	X =  293.358  mm,	Y =   -362.330  mm,	Z =   -225.599  mm,
	W =  0.235 deg,	P =   0.000 deg,	R =   30.000 deg
};
P[726]{
   GP1:
	UF : 0, UT : 6,		CONFIG : 'N U T, 0, 0, 0',
	X =  293.664  mm,	Y =   -361.839  mm,	Z =   -225.016  mm,
	W =  0.235 deg,	P =   0.000 deg,	R =   30.000 deg
};
P[727]{
   GP1:
	UF : 0, UT : 6,		CONFIG : 'N U T, 0, 0, 0',
	X =  293.942  mm,	Y =   -360.846  mm,	Z =   -225.924  mm,
	W =  0.235 deg,	P =   0.000 deg,	R =   30.000 deg
};
P[728]{
   GP1:
	UF : 0, UT : 6,		CONFIG : 'N U T, 0, 0, 0',
	X =  294.171  mm,	Y =   -360.115  mm,	Z =   -225.066  mm,
	W =  0.235 deg,	P =   0.000 deg,	R =   30.000 deg
};
P[729]{
   GP1:
	UF : 0, UT : 6,		CONFIG : 'N U T, 0, 0, 0',
	X =  294.153  mm,	Y =   -359.239  mm,	Z =   -225.885  mm,
	W =  0.235 deg,	P =   0.000 deg,	R =   30.000 deg
};
P[730]{
   GP1:
	UF : 0, UT : 6,		CONFIG : 'N U T, 0, 0, 0',
	X =  293.722  mm,	Y =   -357.104  mm,	Z =   -225.135  mm,
	W =  0.235 deg,	P =   0.000 deg,	R =   30.000 deg
};
P[731]{
   GP1:
	UF : 0, UT : 6,		CONFIG : 'N U T, 0, 0, 0',
	X =  293.309  mm,	Y =   -356.401  mm,	Z =   -225.818  mm,
	W =  0.235 deg,	P =   0.000 deg,	R =   30.000 deg
};
P[732]{
   GP1:
	UF : 0, UT : 6,		CONFIG : 'N U T, 0, 0, 0',
	X =  293.138  mm,	Y =   -356.040  mm,	Z =   -225.356  mm,
	W =  0.235 deg,	P =   0.000 deg,	R =   30.000 deg
};
P[733]{
   GP1:
	UF : 0, UT : 6,		CONFIG : 'N U T, 0, 0, 0',
	X =  292.629  mm,	Y =   -355.102  mm,	Z =   -224.956  mm,
	W =  0.235 deg,	P =   0.000 deg,	R =   30.000 deg
};
P[734]{
   GP1:
	UF : 0, UT : 6,		CONFIG : 'N U T, 0, 0, 0',
	X =  292.218  mm,	Y =   -354.513  mm,	Z =   -225.830  mm,
	W =  0.235 deg,	P =   0.000 deg,	R =   30.000 deg
};
P[735]{
   GP1:
	UF : 0, UT : 6,		CONFIG : 'N U T, 0, 0, 0',
	X =  291.895  mm,	Y =   -353.886  mm,	Z =   -225.347  mm,
	W =  0.235 deg,	P =   0.000 deg,	R =   30.000 deg
};
P[736]{
   GP1:
	UF : 0, UT : 6,		CONFIG : 'N U T, 0, 0, 0',
	X =  291.585  mm,	Y =   -353.345  mm,	Z =   -225.316  mm,
	W =  0.235 deg,	P =   0.000 deg,	R =   30.000 deg
};
P[737]{
   GP1:
	UF : 0, UT : 6,		CONFIG : 'N U T, 0, 0, 0',
	X =  291.141  mm,	Y =   -352.652  mm,	Z =   -225.865  mm,
	W =  0.235 deg,	P =   0.000 deg,	R =   30.000 deg
};
P[738]{
   GP1:
	UF : 0, UT : 6,		CONFIG : 'N U T, 0, 0, 0',
	X =  290.864  mm,	Y =   -352.042  mm,	Z =   -224.936  mm,
	W =  0.235 deg,	P =   0.000 deg,	R =   30.000 deg
};
P[739]{
   GP1:
	UF : 0, UT : 6,		CONFIG : 'N U T, 0, 0, 0',
	X =  290.103  mm,	Y =   -350.838  mm,	Z =   -225.753  mm,
	W =  0.235 deg,	P =   0.000 deg,	R =   30.000 deg
};
P[740]{
   GP1:
	UF : 0, UT : 6,		CONFIG : 'N U T, 0, 0, 0',
	X =  289.640  mm,	Y =   -349.988  mm,	Z =   -225.398  mm,
	W =  0.235 deg,	P =   0.000 deg,	R =   30.000 deg
};
P[741]{
   GP1:
	UF : 0, UT : 6,		CONFIG : 'N U T, 0, 0, 0',
	X =  289.363  mm,	Y =   -349.454  mm,	Z =   -225.022  mm,
	W =  0.235 deg,	P =   0.000 deg,	R =   30.000 deg
};
P[742]{
   GP1:
	UF : 0, UT : 6,		CONFIG : 'N U T, 0, 0, 0',
	X =  288.977  mm,	Y =   -348.910  mm,	Z =   -225.902  mm,
	W =  0.235 deg,	P =   0.000 deg,	R =   30.000 deg
};
P[743]{
   GP1:
	UF : 0, UT : 6,		CONFIG : 'N U T, 0, 0, 0',
	X =  289.007  mm,	Y =   -348.832  mm,	Z =   -224.979  mm,
	W =  0.235 deg,	P =   0.000 deg,	R =   30.000 deg
};
P[744]{
   GP1:
	UF : 0, UT : 6,		CONFIG : 'N U T, 0, 0, 0',
	X =  288.598  mm,	Y =   -348.245  mm,	Z =   -225.836  mm,
	W =  0.235 deg,	P =   0.000 deg,	R =   30.000 deg
};
P[745]{
   GP1:
	UF : 0, UT : 6,		CONFIG : 'N U T, 0, 0, 0',
	X =  287.905  mm,	Y =   -347.052  mm,	Z =   -225.898  mm,
	W =  0.235 deg,	P =   0.000 deg,	R =   30.000 deg
};
P[746]{
   GP1:
	UF : 0, UT : 6,		CONFIG : 'N U T, 0, 0, 0',
	X =  287.856  mm,	Y =   -346.888  mm,	Z =   -225.331  mm,
	W =  0.235 deg,	P =   0.000 deg,	R =   30.000 deg
};
P[747]{
   GP1:
	UF : 0, UT : 6,		CONFIG : 'N U T, 0, 0, 0',
	X =  287.597  mm,	Y =   -346.401  mm,	Z =   -225.057  mm,
	W =  0.235 deg,	P =   0.000 deg,	R =   30.000 deg
};
P[748]{
   GP1:
	UF : 0, UT : 6,		CONFIG : 'N U T, 0, 0, 0',
	X =  287.465  mm,	Y =   -346.283  mm,	Z =   -225.843  mm,
	W =  0.235 deg,	P =   0.000 deg,	R =   30.000 deg
};
P[749]{
   GP1:
	UF : 0, UT : 6,		CONFIG : 'N U T, 0, 0, 0',
	X =  287.067  mm,	Y =   -345.531  mm,	Z =   -225.390  mm,
	W =  0.235 deg,	P =   0.000 deg,	R =   30.000 deg
};
P[750]{
   GP1:
	UF : 0, UT : 6,		CONFIG : 'N U T, 0, 0, 0',
	X =  286.843  mm,	Y =   -345.140  mm,	Z =   -225.369  mm,
	W =  0.235 deg,	P =   0.000 deg,	R =   30.000 deg
};
P[751]{
   GP1:
	UF : 0, UT : 6,		CONFIG : 'N U T, 0, 0, 0',
	X =  286.413  mm,	Y =   -344.462  mm,	Z =   -225.853  mm,
	W =  0.235 deg,	P =   0.000 deg,	R =   30.000 deg
};
P[752]{
   GP1:
	UF : 0, UT : 6,		CONFIG : 'N U T, 0, 0, 0',
	X =  286.421  mm,	Y =   -344.404  mm,	Z =   -225.339  mm,
	W =  0.235 deg,	P =   0.000 deg,	R =   30.000 deg
};
P[753]{
   GP1:
	UF : 0, UT : 6,		CONFIG : 'N U T, 0, 0, 0',
	X =  286.104  mm,	Y =   -343.799  mm,	Z =   -224.934  mm,
	W =  0.235 deg,	P =   0.000 deg,	R =   30.000 deg
};
P[754]{
   GP1:
	UF : 0, UT : 6,		CONFIG : 'N U T, 0, 0, 0',
	X =  285.703  mm,	Y =   -343.227  mm,	Z =   -225.814  mm,
	W =  0.235 deg,	P =   0.000 deg,	R =   30.000 deg
};
P[755]{
   GP1:
	UF : 0, UT : 6,		CONFIG : 'N U T, 0, 0, 0',
	X =  285.716  mm,	Y =   -343.185  mm,	Z =   -225.352  mm,
	W =  0.235 deg,	P =   0.000 deg,	R =   30.000 deg
};
P[756]{
   GP1:
	UF : 0, UT : 6,		CONFIG : 'N U T, 0, 0, 0',
	X =  285.021  mm,	Y =   -342.055  mm,	Z =   -225.883  mm,
	W =  0.235 deg,	P =   0.000 deg,	R =   30.000 deg
};
P[757]{
   GP1:
	UF : 0, UT : 6,		CONFIG : 'N U T, 0, 0, 0',
	X =  285.006  mm,	Y =   -341.909  mm,	Z =   -225.026  mm,
	W =  0.235 deg,	P =   0.000 deg,	R =   30.000 deg
};
P[758]{
   GP1:
	UF : 0, UT : 6,		CONFIG : 'N U T, 0, 0, 0',
	X =  284.638  mm,	Y =   -341.396  mm,	Z =   -225.905  mm,
	W =  0.235 deg,	P =   0.000 deg,	R =   30.000 deg
};
P[759]{
   GP1:
	UF : 0, UT : 6,		CONFIG : 'N U T, 0, 0, 0',
	X =  284.542  mm,	Y =   -341.157  mm,	Z =   -225.390  mm,
	W =  0.235 deg,	P =   0.000 deg,	R =   30.000 deg
};
P[760]{
   GP1:
	UF : 0, UT : 6,		CONFIG : 'N U T, 0, 0, 0',
	X =  284.260  mm,	Y =   -340.728  mm,	Z =   -225.825  mm,
	W =  0.235 deg,	P =   0.000 deg,	R =   30.000 deg
};
P[761]{
   GP1:
	UF : 0, UT : 6,		CONFIG : 'N U T, 0, 0, 0',
	X =  283.947  mm,	Y =   -340.179  mm,	Z =   -225.757  mm,
	W =  0.235 deg,	P =   0.000 deg,	R =   30.000 deg
};
P[762]{
   GP1:
	UF : 0, UT : 6,		CONFIG : 'N U T, 0, 0, 0',
	X =  283.943  mm,	Y =   -340.076  mm,	Z =   -225.084  mm,
	W =  0.235 deg,	P =   0.000 deg,	R =   30.000 deg
};
P[763]{
   GP1:
	UF : 0, UT : 6,		CONFIG : 'N U T, 0, 0, 0',
	X =  283.652  mm,	Y =   -339.616  mm,	Z =   -225.393  mm,
	W =  0.235 deg,	P =   0.000 deg,	R =   30.000 deg
};
P[764]{
   GP1:
	UF : 0, UT : 6,		CONFIG : 'N U T, 0, 0, 0',
	X =  283.491  mm,	Y =   -339.401  mm,	Z =   -225.842  mm,
	W =  0.235 deg,	P =   0.000 deg,	R =   30.000 deg
};
P[765]{
   GP1:
	UF : 0, UT : 6,		CONFIG : 'N U T, 0, 0, 0',
	X =  283.214  mm,	Y =   -338.810  mm,	Z =   -225.058  mm,
	W =  0.235 deg,	P =   0.000 deg,	R =   30.000 deg
};
P[766]{
   GP1:
	UF : 0, UT : 6,		CONFIG : 'N U T, 0, 0, 0',
	X =  283.095  mm,	Y =   -338.710  mm,	Z =   -225.807  mm,
	W =  0.235 deg,	P =   0.000 deg,	R =   30.000 deg
};
P[767]{
   GP1:
	UF : 0, UT : 6,		CONFIG : 'N U T, 0, 0, 0',
	X =  282.884  mm,	Y =   -338.277  mm,	Z =   -225.332  mm,
	W =  0.235 deg,	P =   0.000 deg,	R =   30.000 deg
};
P[768]{
   GP1:
	UF : 0, UT : 6,		CONFIG : 'N U T, 0, 0, 0',
	X =  282.774  mm,	Y =   -338.163  mm,	Z =   -225.876  mm,
	W =  0.235 deg,	P =   0.000 deg,	R =   30.000 deg
};
P[769]{
   GP1:
	UF : 0, UT : 6,		CONFIG : 'N U T, 0, 0, 0',
	X =  282.433  mm,	Y =   -337.456  mm,	Z =   -225.052  mm,
	W =  0.235 deg,	P =   0.000 deg,	R =   30.000 deg
};
P[770]{
   GP1:
	UF : 0, UT : 6,		CONFIG : 'N U T, 0, 0, 0',
	X =  282.371  mm,	Y =   -337.390  mm,	Z =   -225.326  mm,
	W =  0.235 deg,	P =   0.000 deg,	R =   30.000 deg
};
P[771]{
   GP1:
	UF : 0, UT : 6,		CONFIG : 'N U T, 0, 0, 0',
	X =  282.036  mm,	Y =   -336.813  mm,	Z =   -225.375  mm,
	W =  0.235 deg,	P =   0.000 deg,	R =   30.000 deg
};
P[772]{
   GP1:
	UF : 0, UT : 6,		CONFIG : 'N U T, 0, 0, 0',
	X =  281.781  mm,	Y =   -336.317  mm,	Z =   -224.967  mm,
	W =  0.235 deg,	P =   0.000 deg,	R =   30.000 deg
};
P[773]{
   GP1:
	UF : 0, UT : 6,		CONFIG : 'N U T, 0, 0, 0',
	X =  281.391  mm,	Y =   -335.773  mm,	Z =   -225.912  mm,
	W =  0.235 deg,	P =   0.000 deg,	R =   30.000 deg
};
P[774]{
   GP1:
	UF : 0, UT : 6,		CONFIG : 'N U T, 0, 0, 0',
	X =  281.317  mm,	Y =   -335.568  mm,	Z =   -225.365  mm,
	W =  0.235 deg,	P =   0.000 deg,	R =   30.000 deg
};
P[775]{
   GP1:
	UF : 0, UT : 6,		CONFIG : 'N U T, 0, 0, 0',
	X =  281.033  mm,	Y =   -335.035  mm,	Z =   -225.072  mm,
	W =  0.235 deg,	P =   0.000 deg,	R =   30.000 deg
};
P[776]{
   GP1:
	UF : 0, UT : 6,		CONFIG : 'N U T, 0, 0, 0',
	X =  280.601  mm,	Y =   -334.379  mm,	Z =   -225.726  mm,
	W =  0.235 deg,	P =   0.000 deg,	R =   30.000 deg
};
P[777]{
   GP1:
	UF : 0, UT : 6,		CONFIG : 'N U T, 0, 0, 0',
	X =  280.243  mm,	Y =   -333.754  mm,	Z =   -225.695  mm,
	W =  0.235 deg,	P =   0.000 deg,	R =   30.000 deg
};
P[778]{
   GP1:
	UF : 0, UT : 6,		CONFIG : 'N U T, 0, 0, 0',
	X =  279.974  mm,	Y =   -333.246  mm,	Z =   -225.385  mm,
	W =  0.235 deg,	P =   0.000 deg,	R =   30.000 deg
};
P[779]{
   GP1:
	UF : 0, UT : 6,		CONFIG : 'N U T, 0, 0, 0',
	X =  279.552  mm,	Y =   -332.568  mm,	Z =   -225.775  mm,
	W =  0.235 deg,	P =   0.000 deg,	R =   30.000 deg
};
P[780]{
   GP1:
	UF : 0, UT : 6,		CONFIG : 'N U T, 0, 0, 0',
	X =  279.425  mm,	Y =   -332.285  mm,	Z =   -225.323  mm,
	W =  0.235 deg,	P =   0.000 deg,	R =   30.000 deg
};
P[781]{
   GP1:
	UF : 0, UT : 6,		CONFIG : 'N U T, 0, 0, 0',
	X =  279.142  mm,	Y =   -331.800  mm,	Z =   -225.363  mm,
	W =  0.235 deg,	P =   0.000 deg,	R =   30.000 deg
};
P[782]{
   GP1:
	UF : 0, UT : 6,		CONFIG : 'N U T, 0, 0, 0',
	X =  278.831  mm,	Y =   -331.331  mm,	Z =   -225.853  mm,
	W =  0.235 deg,	P =   0.000 deg,	R =   30.000 deg
};
P[783]{
   GP1:
	UF : 0, UT : 6,		CONFIG : 'N U T, 0, 0, 0',
	X =  278.414  mm,	Y =   -330.611  mm,	Z =   -225.873  mm,
	W =  0.235 deg,	P =   0.000 deg,	R =   30.000 deg
};
P[784]{
   GP1:
	UF : 0, UT : 6,		CONFIG : 'N U T, 0, 0, 0',
	X =  278.063  mm,	Y =   -330.063  mm,	Z =   -225.851  mm,
	W =  0.235 deg,	P =   0.000 deg,	R =   30.000 deg
};
P[785]{
   GP1:
	UF : 0, UT : 6,		CONFIG : 'N U T, 0, 0, 0',
	X =  277.652  mm,	Y =   -329.413  mm,	Z =   -224.975  mm,
	W =  0.235 deg,	P =   0.000 deg,	R =   30.000 deg
};
P[786]{
   GP1:
	UF : 0, UT : 6,		CONFIG : 'N U T, 0, 0, 0',
	X =  276.939  mm,	Y =   -328.843  mm,	Z =   -225.875  mm,
	W =  0.235 deg,	P =   0.000 deg,	R =   30.000 deg
};
P[787]{
   GP1:
	UF : 0, UT : 6,		CONFIG : 'N U T, 0, 0, 0',
	X =  276.505  mm,	Y =   -328.450  mm,	Z =   -224.928  mm,
	W =  0.235 deg,	P =   0.000 deg,	R =   30.000 deg
};
P[788]{
   GP1:
	UF : 0, UT : 6,		CONFIG : 'N U T, 0, 0, 0',
	X =  276.052  mm,	Y =   -328.176  mm,	Z =   -224.961  mm,
	W =  0.235 deg,	P =   0.000 deg,	R =   30.000 deg
};
P[789]{
   GP1:
	UF : 0, UT : 6,		CONFIG : 'N U T, 0, 0, 0',
	X =  275.949  mm,	Y =   -328.202  mm,	Z =   -225.686  mm,
	W =  0.235 deg,	P =   0.000 deg,	R =   30.000 deg
};
P[790]{
   GP1:
	UF : 0, UT : 6,		CONFIG : 'N U T, 0, 0, 0',
	X =  275.014  mm,	Y =   -327.801  mm,	Z =   -224.980  mm,
	W =  0.235 deg,	P =   0.000 deg,	R =   30.000 deg
};
P[791]{
   GP1:
	UF : 0, UT : 6,		CONFIG : 'N U T, 0, 0, 0',
	X =  274.857  mm,	Y =   -327.845  mm,	Z =   -225.925  mm,
	W =  0.235 deg,	P =   0.000 deg,	R =   30.000 deg
};
P[792]{
   GP1:
	UF : 0, UT : 6,		CONFIG : 'N U T, 0, 0, 0',
	X =  273.400  mm,	Y =   -327.581  mm,	Z =   -225.074  mm,
	W =  0.235 deg,	P =   0.000 deg,	R =   30.000 deg
};
P[793]{
   GP1:
	UF : 0, UT : 6,		CONFIG : 'N U T, 0, 0, 0',
	X =  273.332  mm,	Y =   -327.624  mm,	Z =   -225.606  mm,
	W =  0.235 deg,	P =   0.000 deg,	R =   30.000 deg
};
P[794]{
   GP1:
	UF : 0, UT : 6,		CONFIG : 'N U T, 0, 0, 0',
	X =  271.568  mm,	Y =   -327.736  mm,	Z =   -224.950  mm,
	W =  0.235 deg,	P =   0.000 deg,	R =   30.000 deg
};
P[795]{
   GP1:
	UF : 0, UT : 6,		CONFIG : 'N U T, 0, 0, 0',
	X =  254.476  mm,	Y =   -350.006  mm,	Z =   -225.113  mm,
	W =  90.000 deg,	P =   -89.765 deg,	R =   30.000 deg
};
P[796]{
   GP1:
	UF : 0, UT : 6,		CONFIG : 'N U T, 0, 0, 0',
	X =  254.492  mm,	Y =   -349.646  mm,	Z =   -224.949  mm,
	W =  90.000 deg,	P =   -89.765 deg,	R =   30.000 deg
};
P[797]{
   GP1:
	UF : 0, UT : 6,		CONFIG : 'N U T, 0, 0, 0',
	X =  254.026  mm,	Y =   -349.246  mm,	Z =   -225.294  mm,
	W =  90.000 deg,	P =   -89.765 deg,	R =   30.000 deg
};
P[798]{
   GP1:
	UF : 0, UT : 6,		CONFIG : 'N U T, 0, 0, 0',
	X =  253.383  mm,	Y =   -349.606  mm,	Z =   -225.773  mm,
	W =  90.000 deg,	P =   -89.765 deg,	R =   30.000 deg
};
P[799]{
   GP1:
	UF : 0, UT : 6,		CONFIG : 'N U T, 0, 0, 0',
	X =  252.761  mm,	Y =   -349.972  mm,	Z =   -225.851  mm,
	W =  90.000 deg,	P =   -89.765 deg,	R =   30.000 deg
};
P[800]{
   GP1:
	UF : 0, UT : 6,		CONFIG : 'N U T, 0, 0, 0',
	X =  252.751  mm,	Y =   -349.908  mm,	Z =   -224.994  mm,
	W =  90.000 deg,	P =   -89.765 deg,	R =   30.000 deg
};
P[801]{
   GP1:
	UF : 0, UT : 6,		CONFIG : 'N U T, 0, 0, 0',
	X =  252.413  mm,	Y =   -350.178  mm,	Z =   -225.923  mm,
	W =  90.000 deg,	P =   -89.765 deg,	R =   30.000 deg
};
P[802]{
   GP1:
	UF : 0, UT : 6,		CONFIG : 'N U T, 0, 0, 0',
	X =  252.163  mm,	Y =   -350.316  mm,	Z =   -225.836  mm,
	W =  90.000 deg,	P =   -89.765 deg,	R =   30.000 deg
};
P[803]{
   GP1:
	UF : 0, UT : 6,		CONFIG : 'N U T, 0, 0, 0',
	X =  251.862  mm,	Y =   -350.423  mm,	Z =   -225.010  mm,
	W =  90.000 deg,	P =   -89.765 deg,	R =   30.000 deg
};
P[804]{
   GP1:
	UF : 0, UT : 6,		CONFIG : 'N U T, 0, 0, 0',
	X =  251.518  mm,	Y =   -350.695  mm,	Z =   -225.921  mm,
	W =  90.000 deg,	P =   -89.765 deg,	R =   30.000 deg
};
P[805]{
   GP1:
	UF : 0, UT : 6,		CONFIG : 'N U T, 0, 0, 0',
	X =  251.231  mm,	Y =   -350.820  mm,	Z =   -225.415  mm,
	W =  90.000 deg,	P =   -89.765 deg,	R =   30.000 deg
};
P[806]{
   GP1:
	UF : 0, UT : 6,		CONFIG : 'N U T, 0, 0, 0',
	X =  250.595  mm,	Y =   -351.225  mm,	Z =   -225.884  mm,
	W =  90.000 deg,	P =   -89.765 deg,	R =   30.000 deg
};
P[807]{
   GP1:
	UF : 0, UT : 6,		CONFIG : 'N U T, 0, 0, 0',
	X =  250.354  mm,	Y =   -351.292  mm,	Z =   -224.994  mm,
	W =  90.000 deg,	P =   -89.765 deg,	R =   30.000 deg
};
P[808]{
   GP1:
	UF : 0, UT : 6,		CONFIG : 'N U T, 0, 0, 0',
	X =  250.275  mm,	Y =   -351.412  mm,	Z =   -225.913  mm,
	W =  90.000 deg,	P =   -89.765 deg,	R =   30.000 deg
};
P[809]{
   GP1:
	UF : 0, UT : 6,		CONFIG : 'N U T, 0, 0, 0',
	X =  250.009  mm,	Y =   -351.490  mm,	Z =   -224.981  mm,
	W =  90.000 deg,	P =   -89.765 deg,	R =   30.000 deg
};
P[810]{
   GP1:
	UF : 0, UT : 6,		CONFIG : 'N U T, 0, 0, 0',
	X =  249.644  mm,	Y =   -351.771  mm,	Z =   -225.845  mm,
	W =  90.000 deg,	P =   -89.765 deg,	R =   30.000 deg
};
P[811]{
   GP1:
	UF : 0, UT : 6,		CONFIG : 'N U T, 0, 0, 0',
	X =  249.076  mm,	Y =   -352.062  mm,	Z =   -225.385  mm,
	W =  90.000 deg,	P =   -89.765 deg,	R =   30.000 deg
};
P[812]{
   GP1:
	UF : 0, UT : 6,		CONFIG : 'N U T, 0, 0, 0',
	X =  248.485  mm,	Y =   -352.369  mm,	Z =   -224.958  mm,
	W =  90.000 deg,	P =   -89.765 deg,	R =   30.000 deg
};
P[813]{
   GP1:
	UF : 0, UT : 6,		CONFIG : 'N U T, 0, 0, 0',
	X =  248.437  mm,	Y =   -352.432  mm,	Z =   -225.404  mm,
	W =  90.000 deg,	P =   -89.765 deg,	R =   30.000 deg
};
P[814]{
   GP1:
	UF : 0, UT : 6,		CONFIG : 'N U T, 0, 0, 0',
	X =  248.192  mm,	Y =   -352.610  mm,	Z =   -225.858  mm,
	W =  90.000 deg,	P =   -89.765 deg,	R =   30.000 deg
};
P[815]{
   GP1:
	UF : 0, UT : 6,		CONFIG : 'N U T, 0, 0, 0',
	X =  248.150  mm,	Y =   -352.559  mm,	Z =   -224.927  mm,
	W =  90.000 deg,	P =   -89.765 deg,	R =   30.000 deg
};
P[816]{
   GP1:
	UF : 0, UT : 6,		CONFIG : 'N U T, 0, 0, 0',
	X =  247.609  mm,	Y =   -352.879  mm,	Z =   -225.011  mm,
	W =  90.000 deg,	P =   -89.765 deg,	R =   30.000 deg
};
P[817]{
   GP1:
	UF : 0, UT : 6,		CONFIG : 'N U T, 0, 0, 0',
	X =  246.915  mm,	Y =   -353.353  mm,	Z =   -225.921  mm,
	W =  90.000 deg,	P =   -89.765 deg,	R =   30.000 deg
};
P[818]{
   GP1:
	UF : 0, UT : 6,		CONFIG : 'N U T, 0, 0, 0',
	X =  246.614  mm,	Y =   -353.516  mm,	Z =   -225.791  mm,
	W =  90.000 deg,	P =   -89.765 deg,	R =   30.000 deg
};
P[819]{
   GP1:
	UF : 0, UT : 6,		CONFIG : 'N U T, 0, 0, 0',
	X =  246.352  mm,	Y =   -353.637  mm,	Z =   -225.414  mm,
	W =  90.000 deg,	P =   -89.765 deg,	R =   30.000 deg
};
P[820]{
   GP1:
	UF : 0, UT : 6,		CONFIG : 'N U T, 0, 0, 0',
	X =  246.063  mm,	Y =   -353.800  mm,	Z =   -225.371  mm,
	W =  90.000 deg,	P =   -89.765 deg,	R =   30.000 deg
};
P[821]{
   GP1:
	UF : 0, UT : 6,		CONFIG : 'N U T, 0, 0, 0',
	X =  245.719  mm,	Y =   -354.039  mm,	Z =   -225.870  mm,
	W =  90.000 deg,	P =   -89.765 deg,	R =   30.000 deg
};
P[822]{
   GP1:
	UF : 0, UT : 6,		CONFIG : 'N U T, 0, 0, 0',
	X =  245.407  mm,	Y =   -354.219  mm,	Z =   -225.868  mm,
	W =  90.000 deg,	P =   -89.765 deg,	R =   30.000 deg
};
P[823]{
   GP1:
	UF : 0, UT : 6,		CONFIG : 'N U T, 0, 0, 0',
	X =  244.785  mm,	Y =   -354.579  mm,	Z =   -225.878  mm,
	W =  90.000 deg,	P =   -89.765 deg,	R =   30.000 deg
};
P[824]{
   GP1:
	UF : 0, UT : 6,		CONFIG : 'N U T, 0, 0, 0',
	X =  244.493  mm,	Y =   -354.751  mm,	Z =   -225.915  mm,
	W =  90.000 deg,	P =   -89.765 deg,	R =   30.000 deg
};
P[825]{
   GP1:
	UF : 0, UT : 6,		CONFIG : 'N U T, 0, 0, 0',
	X =  244.186  mm,	Y =   -354.850  mm,	Z =   -224.944  mm,
	W =  90.000 deg,	P =   -89.765 deg,	R =   30.000 deg
};
P[826]{
   GP1:
	UF : 0, UT : 6,		CONFIG : 'N U T, 0, 0, 0',
	X =  243.580  mm,	Y =   -355.277  mm,	Z =   -225.903  mm,
	W =  90.000 deg,	P =   -89.765 deg,	R =   30.000 deg
};
P[827]{
   GP1:
	UF : 0, UT : 6,		CONFIG : 'N U T, 0, 0, 0',
	X =  243.552  mm,	Y =   -355.219  mm,	Z =   -224.989  mm,
	W =  90.000 deg,	P =   -89.765 deg,	R =   30.000 deg
};
P[828]{
   GP1:
	UF : 0, UT : 6,		CONFIG : 'N U T, 0, 0, 0',
	X =  243.238  mm,	Y =   -355.460  mm,	Z =   -225.728  mm,
	W =  90.000 deg,	P =   -89.765 deg,	R =   30.000 deg
};
P[829]{
   GP1:
	UF : 0, UT : 6,		CONFIG : 'N U T, 0, 0, 0',
	X =  242.979  mm,	Y =   -355.552  mm,	Z =   -225.015  mm,
	W =  90.000 deg,	P =   -89.765 deg,	R =   30.000 deg
};
P[830]{
   GP1:
	UF : 0, UT : 6,		CONFIG : 'N U T, 0, 0, 0',
	X =  242.821  mm,	Y =   -355.673  mm,	Z =   -225.377  mm,
	W =  90.000 deg,	P =   -89.765 deg,	R =   30.000 deg
};
P[831]{
   GP1:
	UF : 0, UT : 6,		CONFIG : 'N U T, 0, 0, 0',
	X =  242.654  mm,	Y =   -355.811  mm,	Z =   -225.897  mm,
	W =  90.000 deg,	P =   -89.765 deg,	R =   30.000 deg
};
P[832]{
   GP1:
	UF : 0, UT : 6,		CONFIG : 'N U T, 0, 0, 0',
	X =  242.346  mm,	Y =   -355.915  mm,	Z =   -224.979  mm,
	W =  90.000 deg,	P =   -89.765 deg,	R =   30.000 deg
};
P[833]{
   GP1:
	UF : 0, UT : 6,		CONFIG : 'N U T, 0, 0, 0',
	X =  241.135  mm,	Y =   -356.678  mm,	Z =   -225.767  mm,
	W =  90.000 deg,	P =   -89.765 deg,	R =   30.000 deg
};
P[834]{
   GP1:
	UF : 0, UT : 6,		CONFIG : 'N U T, 0, 0, 0',
	X =  240.535  mm,	Y =   -357.031  mm,	Z =   -225.858  mm,
	W =  90.000 deg,	P =   -89.765 deg,	R =   30.000 deg
};
P[835]{
   GP1:
	UF : 0, UT : 6,		CONFIG : 'N U T, 0, 0, 0',
	X =  240.184  mm,	Y =   -357.234  mm,	Z =   -225.858  mm,
	W =  90.000 deg,	P =   -89.765 deg,	R =   30.000 deg
};
P[836]{
   GP1:
	UF : 0, UT : 6,		CONFIG : 'N U T, 0, 0, 0',
	X =  239.890  mm,	Y =   -357.329  mm,	Z =   -224.933  mm,
	W =  90.000 deg,	P =   -89.765 deg,	R =   30.000 deg
};
P[837]{
   GP1:
	UF : 0, UT : 6,		CONFIG : 'N U T, 0, 0, 0',
	X =  239.840  mm,	Y =   -357.435  mm,	Z =   -225.888  mm,
	W =  90.000 deg,	P =   -89.765 deg,	R =   30.000 deg
};
P[838]{
   GP1:
	UF : 0, UT : 6,		CONFIG : 'N U T, 0, 0, 0',
	X =  239.597  mm,	Y =   -357.578  mm,	Z =   -225.914  mm,
	W =  90.000 deg,	P =   -89.765 deg,	R =   30.000 deg
};
P[839]{
   GP1:
	UF : 0, UT : 6,		CONFIG : 'N U T, 0, 0, 0',
	X =  239.239  mm,	Y =   -357.771  mm,	Z =   -225.755  mm,
	W =  90.000 deg,	P =   -89.765 deg,	R =   30.000 deg
};
P[840]{
   GP1:
	UF : 0, UT : 6,		CONFIG : 'N U T, 0, 0, 0',
	X =  238.979  mm,	Y =   -357.891  mm,	Z =   -225.378  mm,
	W =  90.000 deg,	P =   -89.765 deg,	R =   30.000 deg
};
P[841]{
   GP1:
	UF : 0, UT : 6,		CONFIG : 'N U T, 0, 0, 0',
	X =  238.623  mm,	Y =   -358.136  mm,	Z =   -225.867  mm,
	W =  90.000 deg,	P =   -89.765 deg,	R =   30.000 deg
};
P[842]{
   GP1:
	UF : 0, UT : 6,		CONFIG : 'N U T, 0, 0, 0',
	X =  238.325  mm,	Y =   -358.239  mm,	Z =   -225.019  mm,
	W =  90.000 deg,	P =   -89.765 deg,	R =   30.000 deg
};
P[843]{
   GP1:
	UF : 0, UT : 6,		CONFIG : 'N U T, 0, 0, 0',
	X =  238.318  mm,	Y =   -358.313  mm,	Z =   -225.868  mm,
	W =  90.000 deg,	P =   -89.765 deg,	R =   30.000 deg
};
P[844]{
   GP1:
	UF : 0, UT : 6,		CONFIG : 'N U T, 0, 0, 0',
	X =  237.729  mm,	Y =   -358.654  mm,	Z =   -225.883  mm,
	W =  90.000 deg,	P =   -89.765 deg,	R =   30.000 deg
};
P[845]{
   GP1:
	UF : 0, UT : 6,		CONFIG : 'N U T, 0, 0, 0',
	X =  237.335  mm,	Y =   -358.843  mm,	Z =   -225.406  mm,
	W =  90.000 deg,	P =   -89.765 deg,	R =   30.000 deg
};
P[846]{
   GP1:
	UF : 0, UT : 6,		CONFIG : 'N U T, 0, 0, 0',
	X =  237.177  mm,	Y =   -358.897  mm,	Z =   -224.947  mm,
	W =  90.000 deg,	P =   -89.765 deg,	R =   30.000 deg
};
P[847]{
   GP1:
	UF : 0, UT : 6,		CONFIG : 'N U T, 0, 0, 0',
	X =  237.096  mm,	Y =   -359.020  mm,	Z =   -225.901  mm,
	W =  90.000 deg,	P =   -89.765 deg,	R =   30.000 deg
};
P[848]{
   GP1:
	UF : 0, UT : 6,		CONFIG : 'N U T, 0, 0, 0',
	X =  236.510  mm,	Y =   -359.289  mm,	Z =   -225.036  mm,
	W =  90.000 deg,	P =   -89.765 deg,	R =   30.000 deg
};
P[849]{
   GP1:
	UF : 0, UT : 6,		CONFIG : 'N U T, 0, 0, 0',
	X =  236.258  mm,	Y =   -359.462  mm,	Z =   -225.381  mm,
	W =  90.000 deg,	P =   -89.765 deg,	R =   30.000 deg
};
P[850]{
   GP1:
	UF : 0, UT : 6,		CONFIG : 'N U T, 0, 0, 0',
	X =  235.905  mm,	Y =   -359.705  mm,	Z =   -225.865  mm,
	W =  90.000 deg,	P =   -89.765 deg,	R =   30.000 deg
};
P[851]{
   GP1:
	UF : 0, UT : 6,		CONFIG : 'N U T, 0, 0, 0',
	X =  235.867  mm,	Y =   -359.653  mm,	Z =   -224.941  mm,
	W =  90.000 deg,	P =   -89.765 deg,	R =   30.000 deg
};
P[852]{
   GP1:
	UF : 0, UT : 6,		CONFIG : 'N U T, 0, 0, 0',
	X =  235.623  mm,	Y =   -359.863  mm,	Z =   -225.803  mm,
	W =  90.000 deg,	P =   -89.765 deg,	R =   30.000 deg
};
P[853]{
   GP1:
	UF : 0, UT : 6,		CONFIG : 'N U T, 0, 0, 0',
	X =  235.230  mm,	Y =   -360.022  mm,	Z =   -224.967  mm,
	W =  90.000 deg,	P =   -89.765 deg,	R =   30.000 deg
};
P[854]{
   GP1:
	UF : 0, UT : 6,		CONFIG : 'N U T, 0, 0, 0',
	X =  234.945  mm,	Y =   -360.189  mm,	Z =   -224.993  mm,
	W =  90.000 deg,	P =   -89.765 deg,	R =   30.000 deg
};
P[855]{
   GP1:
	UF : 0, UT : 6,		CONFIG : 'N U T, 0, 0, 0',
	X =  225.565  mm,	Y =   -342.543  mm,	Z =   -225.473  mm,
	W =  90.000 deg,	P =   0.000 deg,	R =   30.000 deg
};
P[856]{
   GP1:
	UF : 0, UT : 6,		CONFIG : 'N U T, 0, 0, 0',
	X =  240.000  mm,	Y =   -370.000  mm,	Z =   -170.000  mm,
	W =  90.000 deg,	P =   0.000 deg,	R =   30.000 deg
};
/END
